# B&R Automation Studio project RS15_RX_30005_r00 (part 5)

#### A1_Control.var - Local variables
```iecst
(********************************************************************
 * COPYRIGHT -- Microsoft
 ********************************************************************
 * Program: A1_Control
 * File: A1_Control.var
 * Author: pkiel
 * Created: July 12, 2011
 ********************************************************************
 * Local variables of program A1_Control
 ********************************************************************)
VAR
  HGW_ChangeReal_0 : HGW_ChangeReal;
  H_RelativeChangeLimitReal1_0 : H_FB_RelativeChangeLimitReal1 ;
  HGW_Toggle_0 : HGW_Toggle;
  HGW_Toggle_1 : HGW_Toggle;
  HMI_FasterPB : BOOL;
  HMI_SlowerPB : BOOL;
  Synch_Permissive : BOOL;
  TOF_0 : TOF;
  bCmd_ManuTimSetPlus  : BOOL ;
  bCmd_ManuTimSetMoins : BOOL ;
  rTemp_ : ARRAY[0..9] OF REAL ;
  rIncrOffsetAxeRun_Inch : REAL ;

  bManuTimSetCond : BOOL ;
  bShiftPerfPos : BOOL ;
  bShiftPerfNeg : BOOL ;
  bEventSelEnvB : BOOL ;

END_VAR
```

- Program Logical/BagMachine_Section/Perf/Axis1/A1_Automat (IEC) - Cam Automat (no source held here)

### Program Logical/BagMachine_Section/Perf/Axis1/A1_Automat2 (IEC) - Cam Automat For Parking Axis

#### A1_Automat2Cyclic.st
```iecst
(********************************************************************
 * COPYRIGHT -- Microsoft
 ********************************************************************
 * Program: A1_Automat2
 * File: A1_Automat2Cyclic.st
 * Author: pkiel
 * Created: July 19, 2011
 ********************************************************************
 * Implementation of program A1_Automat2
 ********************************************************************)

PROGRAM _CYCLIC

(**** CAM AUTOMAT FOR PARKING AXIS ****)
(**** Initialize Automat Parameters Upon Automat Start Request ****)
	Synch_Request := gPerf_ParkRequest;
	IF (Synch_Request AND NOT ParID_Ready) THEN
		MC_BR_InitMasterParIDTransfer_0.Master:=gA[11].Ident;
	    MC_BR_InitMasterParIDTransfer_0.Slave:=gA[1].Ident;
	    MC_BR_InitMasterParIDTransfer_0.MasterParID:=412;
	    MC_BR_InitMasterParIDTransfer_0.SlaveChannel:=0;
	    MC_BR_InitMasterParIDTransfer_0.Execute:=TRUE;
	    IF (MC_BR_InitMasterParIDTransfer_0.Done) THEN
	      MasterParID:=MC_BR_InitMasterParIDTransfer_0.ReceiveParID;
	      MC_BR_InitMasterParIDTransfer_0.Execute:=FALSE;
	      ParID_Ready:=1;
	    ELSIF (MC_BR_InitMasterParIDTransfer_0.Error) THEN
	    (*Store ErrorID in a variable,
	      ErrorID is reset on falling edge of 'Execute'*)
	      ErrorID:=MC_BR_InitMasterParIDTransfer_0.ErrorID;
	      ParID_Ready:=0;
	      MC_BR_InitMasterParIDTransfer_0.Execute:=FALSE;
	    END_IF
	END_IF
	MC_BR_InitMasterParIDTransfer_0();

(**** Initialize Automat Parameters Upon Automat Start Request ****)
  bInitCamAuto := ParID_Ready    AND
                  g_bCameProf_OK AND
                  1              ;

	IF (EDGEPOS(bInitCamAuto))THEN

		(*general automat parameter*)
			AutData.MasterParID		    := MasterParID;
			AutData.StartPosition		:= 0;
			AutData.StartInterval		:= gA[11].AxisPeriod;
			AutData.MaxMasterVelocity	:= gr_rMachMaxSpeed_BPM ;

		(**** Calculations ****)
			gA[1].InchPerDeg := gA[1].UnitsPerDeg/gA[1].UnitsPerInch;
			Travel_Deg := gSP_A[1].ParkPosition-gSP_A[1].MatchedSpeed;
			IF (Travel_Deg<0) THEN
				Travel_Deg := Travel_Deg+360.0;
			END_IF
			Travel_Inch := Travel_Deg*gA[1].InchPerDeg;
			MatchedSpeed_Inch := gSP_A[1].MatchedSpeed*gA[1].InchPerDeg;
			MasterOffset := 0(*gRecipeActive.Perf_Offset*);
			Slave_AxisPeriod := gA[1].AxisPeriod/gSP_PerfKnifeCount;
      rSlave_AxisPeriod_Inch := Slave_AxisPeriod / gA[1].UnitsPerInch ;
      rPosOutMatchedSpeed2_Inch := MatchedSpeed_Inch + rSlave_AxisPeriod_Inch ;

		(**** Slave Starting In Matched Speed Zone ****)
      IF g_bPerfInMatchedSpeed THEN
        InMatched := 1;

			(*Automat STATE 0 Basis State*)
				AutData.State[0].Event[0].Type		:= ncST_END;
				AutData.State[0].Event[0].Attribute	:= ncAT_ONCE;
        AutData.State[0].Event[0].NextState  := 1;

      rTempPosA1_Inch := H_FC_Modulus(IN_rMod:=360*gA[1].InchPerDeg/gSP_PerfKnifeCount, IN_rVar:=gA[1].PositionInch) ;

			(*Initial Matched Speed Zone*)
				AutData.State[1].CamProfileIndex	:= 16#FFFF;
				AutData.State[1].MasterFactor		:= REAL_TO_UDINT((MatchedSpeed_Inch-rTempPosA1_Inch)*gA[11].UnitsPerInch);
				AutData.State[1].SlaveFactor		:= REAL_TO_DINT((MatchedSpeed_Inch-rTempPosA1_Inch)*gA[1].UnitsPerInch);
				AutData.State[1].CompMode			:= ncOFF;

				AutData.State[1].Event[0].Type		:= ncST_END;
				AutData.State[1].Event[0].Attribute	:= ncST_END;
				AutData.State[1].Event[0].NextState	:= 2;

			(*Initial Comp With Matched Speed Zone*)
				AutData.State[2].CamProfileIndex	:= 16#FFFF;
				AutData.State[2].MasterFactor		:= REAL_TO_UDINT(MatchedSpeed_Inch*gA[11].UnitsPerInch);
				AutData.State[2].SlaveFactor		:= REAL_TO_DINT(MatchedSpeed_Inch*gA[1].UnitsPerInch);
				AutData.State[2].CompMode			:= ncONLYCOMP;
				AutData.State[2].MasterCompDistance	:= (gA[11].AxisPeriod)-((gA[11].PositionInch+MasterOffset)*gA[11].UnitsPerInch)-AutData.State[1].MasterFactor;
				AutData.State[2].SlaveCompDistance	:= (Slave_AxisPeriod)-gA[1].PositionCount-AutData.State[1].SlaveFactor;

				IF (AutData.State[2].SlaveCompDistance<=0) THEN
					AutData.State[2].SlaveCompDistance := AutData.State[2].SlaveCompDistance+Slave_AxisPeriod;
				END_IF
				IF (AutData.State[2].MasterCompDistance<0) THEN
					Value1 := REAL_TO_DINT(AutData.State[2].MasterCompDistance*1000.0);
					Value2 := REAL_TO_DINT(gA[11].AxisPeriod*1000.0);
					AutData.State[2].MasterCompDistance := (DINT_TO_REAL(Value1 MOD Value2))/1000.0;
					IF (AutData.State[2].MasterCompDistance<0) THEN
						AutData.State[2].MasterCompDistance := AutData.State[2].MasterCompDistance+gA[11].AxisPeriod;
					END_IF
				END_IF
				IF ((AutData.State[2].MasterCompDistance<(0.5*gA[11].AxisPeriod)) AND (AutData.State[2].SlaveCompDistance>(0.5*Slave_AxisPeriod))) THEN
					AutData.State[2].MasterCompDistance := AutData.State[2].MasterCompDistance+(gA[11].AxisPeriod);
				END_IF
				IF (AutData.State[2].MasterCompDistance<(0.1*gA[11].AxisPeriod)) THEN
					AutData.State[2].MasterCompDistance := AutData.State[2].MasterCompDistance+(gA[11].AxisPeriod);
				END_IF

				AutData.State[2].Event[0].Type		:= ncST_END;
				AutData.State[2].Event[0].Attribute	:= ncST_END;
				AutData.State[2].Event[0].NextState	:= 3;

			ELSE
				InMatched := 0;

			(*Automat STATE 0 Basis State*)
				AutData.State[0].Event[0].Type		:= ncST_END;
				AutData.State[0].Event[0].Attribute	:= ncAT_ONCE;
				AutData.State[0].Event[0].NextState	:= 2;

			(*Initial Matched Speed Zone...NOT USED*)
				AutData.State[1].CamProfileIndex	:= 16#FFFE;
				AutData.State[1].MasterFactor		:= 1;
				AutData.State[1].SlaveFactor		:= 1;
				AutData.State[1].CompMode			:= ncOFF;

				AutData.State[1].Event[0].Type		:= ncST_END;
				AutData.State[1].Event[0].Attribute	:= ncST_END;
				AutData.State[1].Event[0].NextState	:= 3;

			(*Initial Comp With Matched Speed Zone*)
				AutData.State[2].CamProfileIndex	:= 16#FFFF;
				AutData.State[2].MasterFactor		:= REAL_TO_UDINT(MatchedSpeed_Inch*gA[11].UnitsPerInch);
				AutData.State[2].SlaveFactor		:= REAL_TO_DINT(MatchedSpeed_Inch*gA[1].UnitsPerInch);
				AutData.State[2].CompMode			:= ncONLYCOMP;
				AutData.State[2].MasterCompDistance	:= gA[11].AxisPeriod-((gA[11].PositionInch+MasterOffset)*gA[11].UnitsPerInch);
				AutData.State[2].SlaveCompDistance	:= Slave_AxisPeriod-gA[1].PositionCount;

				IF (AutData.State[2].SlaveCompDistance<=0) THEN
					AutData.State[2].SlaveCompDistance := AutData.State[2].SlaveCompDistance+Slave_AxisPeriod;
				END_IF
				IF (AutData.State[2].MasterCompDistance<0) THEN
					Value1 := REAL_TO_DINT(AutData.State[2].MasterCompDistance*1000.0);
					Value2 := REAL_TO_DINT(gA[11].AxisPeriod*1000.0);
					AutData.State[2].MasterCompDistance := (DINT_TO_REAL(Value1 MOD Value2))/1000.0;
					IF (AutData.State[2].MasterCompDistance<0) THEN
						AutData.State[2].MasterCompDistance := AutData.State[2].MasterCompDistance+gA[11].AxisPeriod;
					END_IF
				END_IF
				IF ((AutData.State[2].MasterCompDistance<(0.5*gA[11].AxisPeriod)) AND (AutData.State[2].SlaveCompDistance>(0.5*Slave_AxisPeriod))) THEN
					AutData.State[2].MasterCompDistance := AutData.State[2].MasterCompDistance+(gA[11].AxisPeriod);
				END_IF
				IF (AutData.State[2].MasterCompDistance<(0.1*gA[11].AxisPeriod)) THEN
					AutData.State[2].MasterCompDistance := AutData.State[2].MasterCompDistance+(gA[11].AxisPeriod);
				END_IF

				AutData.State[2].Event[0].Type		:= ncST_END;
				AutData.State[2].Event[0].Attribute	:= ncST_END;
				AutData.State[2].Event[0].NextState	:= 3;

			END_IF

		(*Running Comp With Matched Speed Zone *)
			AutData.State[3].CamProfileIndex	:= 16#FFFE;
			AutData.State[3].MasterFactor		:= 1;
			AutData.State[3].SlaveFactor		:= 0;
			AutData.State[3].CompMode			:= ncONLYCOMP;
			AutData.State[3].MasterCompDistance	:= Travel_Inch*gA[11].UnitsPerInch;
			AutData.State[3].SlaveCompDistance	:= Travel_Inch*gA[1].UnitsPerInch;

			AutData.State[3].Event[0].Type		:= ncST_END;
			AutData.State[3].Event[0].Attribute	:= ncST_END;
			AutData.State[3].Event[0].NextState	:= 4;

		(*Running Comp With Matched Speed Zone *)
			AutData.State[4].CamProfileIndex	:= 16#FFFF;
			AutData.State[4].MasterFactor		:= REAL_TO_UDINT(Slave_AxisPeriod);
			AutData.State[4].SlaveFactor		:= 0;
			AutData.State[4].CompMode			:= ncOFF;

			AutData.State[4].Event[0].Type		:= ncST_END;
			AutData.State[4].Event[0].Attribute	:= ncST_END;
			AutData.State[4].Event[0].NextState	:= 4;

		(*Initialize & Enable the Automat Control *)
			MC_BR_AutControl_0.Enable 		:= 1;
			MC_BR_AutControl_0.AdrAutData 	:= ADR(AutData);
			MC_BR_AutControl_0.InitAutData 	:= 1;
	END_IF
		(* wait for initialization done*)
			IF ((MC_BR_AutControl_0.AutDataInitialized = 1) AND (Synch_Request)) THEN
				MC_BR_AutControl_0.InitAutData 	:= 0;
				AutomatStart := 1;
			END_IF
			(* check if error occured *)
			IF (MC_BR_AutControl_0.ErrorID <> 0) THEN
				Error := MC_BR_AutControl_0.ErrorID;
				MC_BR_AutControl_0.Enable := 0;
			END_IF

	(******************** ENABLE CAM-AUTOMAT **********************)

	IF (AutomatStart) THEN
			MC_BR_AutControl_0.Start := 1;
			AutomatStart := 0;
	END_IF

	IF (NOT Synch_Request) THEN
			MC_BR_AutControl_0.Stop := 1;
			MC_BR_AutControl_0.Start := 0;
			ParID_Ready := 0;
			IF (MC_BR_AutControl_0.Running=0) THEN
				MC_BR_AutControl_0.Enable := 0;
				MC_BR_AutControl_0.Stop := 0;
			END_IF
	END_IF

	IF (gPerf_ParkRequired) THEN
		gA[1].Ind_AutomatEnabled:=MC_BR_AutControl_0.Enable;
		gA[1].Ind_CurrentAutomatState:=MC_BR_AutControl_0.ActualStateIndex;
	END_IF

	(********************** MC_AUTCONTROL *************************)
	MC_BR_AutControl_0.Slave:= gA[1].Ident;
	MC_BR_AutControl_0();

END_PROGRAM
```

### Program Logical/BagMachine_Section/Perf/Axis1/A1_Ref (IEC) - Reference Routine

#### A1_Ref.var - Local variables
```iecst
(********************************************************************
 * COPYRIGHT -- Microsoft
 ********************************************************************
 * Program: A1_Ref
 * File: A1_Ref.var
 * Author: pkiel
 * Created: July 13, 2011
 ********************************************************************
 * Local variables of program A1_Ref
 ********************************************************************)
VAR
	HGW_2StateIND_0 : HGW_2StateIND;
	HGW_2StepMove_0 : HGW_2StepMove;
	MC_Home_0 : MC_Home;
	RefPBColor_Ind : UINT;
END_VAR
```

### Program Logical/BagMachine_Section/Perf/Axis1/A1_Cycle (IEC) - A new program

#### A1_CycleCyclic.st
```iecst
(********************************************************************
 * COPYRIGHT -- .
 ********************************************************************
 * Program: A1_Cycle
 * File: A1_CycleCyclic.st
 * Author: dominique
 * Created: August 01, 2011
 ********************************************************************
 * Implementation of program A1_Cycle
 ********************************************************************)

PROGRAM _CYCLIC

// Manu axis movement for timing setting

    //---------------------------------------------------------------------------------------------------------------------
    // ACDC Power Supply cycle
    //---------------------------------------------------------------------------------------------------------------------
    // Start cycle
    gstCycA[1].CycManTimSet.CmdStart := ( gA[1].Cmd_ManuTimSetPlus    OR
                                          gA[1].Cmd_ManuTimSetMinus ) AND
                                        NOT(gA[1].Error)              AND
                                        NOT(gA[11].Error)             ;
    IF gstCycA[1].CycManTimSet.CmdStart THEN
      gstCycA[1].CycManTimSet.bSCyc := 1 ;
    END_IF ;

    //----------------------------------------------------------------------
    // Cycle at rest
    IF NOT(gstCycA[1].CycManTimSet.bSCyc) AND
       1                                 THEN
      IF NOT( gstCycA[1].CycManTimSet.bFCyc ) THEN
        // Init after cycle unpropaly ended
        gstCycA[1].CycManTimSet.bFCyc := 1 ;
        gstCycA[1].CycManTimSet.bCyc  := 0 ;

        gstCycA[1].CycManTimSet.CmdMov  := 0 ;
        gstCycA[1].CycManTimSet.CmdStop := 0 ;
        gstCycA[1].CycManTimSet.CmdSynchroOn := 0 ;
      END_IF
      gstCycA[1].CycManTimSet.iStep := 0 ;
      RETURN ;
    ELSE
    //----------------------------------------------------------------------
    // Cycle running

      // Permanent conditions
      IF NOT(gA[1].Ind_Ready)                  OR
         NOT(gA[11].Ind_Ready)                 OR
         NOT(gstCycA[1].CycManTimSet.CmdStart) AND
         (gstCycA[1].CycManTimSet.iStep <= 2)  THEN
        gstCycA[1].CycManTimSet.bSCyc := 0 ;
        RETURN ;
      END_IF

      // Permanent actions
      stTON_01 (
            IN := ( gstCycA[1].CycManTimSet.iStep = C_iSTEP_0 ) ,
            PT := T#30ms
               ) ;
    END_IF
    //----------------------------------------------------------------------
    // Cycle steps

        CASE gstCycA[1].CycManTimSet.iStep OF

        C_iSTEP_0 :
         //----------------------------------------------
         // Etape 1 : Initialisation
         //----------------------------------------------
          IF stTON_01.Q THEN
            gstCycA[1].CycManTimSet.iStep := C_iSTEP_1 ;

            // Action Step 1
            gstCycA[1].CycManTimSet.bFCyc := 0 ;
            gstCycA[1].CycManTimSet.bCyc  := 1 ;
          END_IF

        C_iSTEP_1 :
         //----------------------------------------------
         // Etape 2 : Synchro Drum
         //----------------------------------------------
          IF TRUE THEN
            gstCycA[1].CycManTimSet.iStep := C_iSTEP_2 ;

            // Action Step 2
            gstCycA[1].CycManTimSet.CmdSynchroOn := 1 ;
          END_IF

        C_iSTEP_2 :
         //----------------------------------------------
         // Step 3 : Activation motion and Stop waiting
         //----------------------------------------------
          IF gstCycA[1].CycManTimSet.bSynchroOkSlavA[11] THEN
            gstCycA[1].CycManTimSet.iStep := C_iSTEP_3 ;

            // Action Step 3
            gstCycA[1].CycManTimSet.CmdMov  := 1 ;
            gstCycA[1].CycManTimSet.CmdStop := 0 ;
            // Stop waiting
          END_IF

        C_iSTEP_3 :
         //----------------------------------------------
         // Step 4 : Stop motion and End stop waiting
         //----------------------------------------------
          IF NOT(gstCycA[1].CycManTimSet.CmdStart) THEN
            gstCycA[1].CycManTimSet.iStep := C_iSTEP_4 ;

            // Action Step 4
            gstCycA[1].CycManTimSet.CmdMov  := 0 ;
            gstCycA[1].CycManTimSet.CmdStop := 1 ;
            // End stop waiting
          END_IF

        C_iSTEP_4 :
         //----------------------------------------------
         // Step 3 : Activation motion and Stop waiting
         // Step 5 : Cut synchro
         //----------------------------------------------
          // Condition Step3
          IF gstCycA[1].CycManTimSet.CmdStart THEN
            gstCycA[1].CycManTimSet.iStep := C_iSTEP_3 ;

            // Action Step 3
            gstCycA[1].CycManTimSet.CmdMov  := 1 ;
            gstCycA[1].CycManTimSet.CmdStop := 0 ;
            // Stop waiting
            RETURN ;
          END_IF ;
          // Condition Step5
          IF NOT(gstCycA[1].CycManTimSet.CmdStop) THEN
            gstCycA[1].CycManTimSet.iStep := C_iSTEP_5 ;

            // Action Step 5
            gstCycA[1].CycManTimSet.CmdSynchroOn := 0 ;
          END_IF

        C_iSTEP_5 :
         //----------------------------------------------
         // Step 6 : New offset calculation
         //----------------------------------------------
          IF TRUE THEN
            gstCycA[1].CycManTimSet.iStep := C_iSTEP_6 ;

            // Action Step 6
            // Memo Actual phase Offset
            rTempActPhasDeg[1]    := gRecipeActive.rPerf_PhasMasterDeg ;
            rTempActOffsetInch[1] := gRecipeActive.Perf_Offset ;
            // Update phase
            gRecipeActive.rPerf_PhasMasterDeg := gA[11].rActPhasDeg ;
            // Update Offset
            rTemp_[1] := gA[11].PositionInch - gA[9].PositionInch ;
            gRecipeActive.Perf_Offset := H_FC_Modulus (IN_rMod := gRecipeActive.Repeat, IN_rVar := rTemp_[1]) ;
          END_IF

        C_iSTEP_6 :
         //----------------------------------------------
         // Step 0 : First step
         //----------------------------------------------
          IF TRUE THEN
            gstCycA[1].CycManTimSet.iStep := C_iSTEP_0 ;

            // Action Step 0
            gstCycA[1].CycManTimSet.bSCyc := 0 ;
            gstCycA[1].CycManTimSet.bFCyc := 1 ;
            gstCycA[1].CycManTimSet.bCyc  := 0 ;
          END_IF
        END_CASE
    //---------------------------------------------------------------------------------------------------------------------

END_PROGRAM
```

### Program Logical/BagMachine_Section/Perf/Axis1/A1_CamProfCalc (IEC) - A new program

#### A1_CamProfCalcInit.st - Initialization code
```iecst
(********************************************************************
 * COPYRIGHT -- .
 ********************************************************************
 * Program: A1_CamProfCalc
 * File: A1_CamProfCalcInit.st
 * Author: dominique
 * Created: August 24, 2011
 ********************************************************************
 * Implementation of program A1_CamProfCalc
 ********************************************************************)

PROGRAM _INIT
  // Came profile Perf index
  g_uiIndexCamProfPerf := 1 ;

END_PROGRAM
```

### Program Logical/BagMachine_Section/Perf/Axis11_VirtualAxis/A11_Automat

#### A11_AutomatCyclic.st
```iecst
(********************************************************************
 * COPYRIGHT -- Microsoft
 ********************************************************************
 * Program: A11_Automat
 * File: A11_AutomatCyclic.st
 * Author: pkiel
 * Created: July 22, 2011
 ********************************************************************
 * Implementation of program A11_Automat
 ********************************************************************)

PROGRAM _CYCLIC

  // Synchro ratio Master/Slave
     // Master = Virtuel
     gA[11].rRSynNum := 1 ;
     gA[11].rRSynDen := 1 ;

  // Signal synchro Holding axis
  MC_BR_AutControl_0.Signal1 := gA[3].Ind_bSynchroOK ;

  // Perf  manu moving
  MC_BR_AutControl_0.Signal2 := 0 ;

  IF gstCycA[1].CycManTimSet.CmdSynchroOn THEN
    MC_BR_AutControl_0.Signal2 := 1 ;
  END_IF

  // A11 Synchro OK indicator
  gstCycA[1].CycManTimSet.bSynchroOkSlavA[11] := ( MC_BR_AutControl_0.ActualStateIndex = 3 )   AND
                                                 gA[11].Ind_SynchronizedMotion AND ParID_Ready ;

(**** STRAIGHT GEARED CAM AUTOMAT WITH ABSOLUTE PHASE SYNCHRONIZATION FOR TEARING AXIS ***)

(* Set Up Master Position Parameter ID *)
  Synch_Request := gA[11].Cmd_SynchronizedMotion;
  IF (Synch_Request AND NOT ParID_Ready) THEN
    MC_BR_InitMasterParIDTransfer_0.Master:=gA[9].Ident;
      MC_BR_InitMasterParIDTransfer_0.Slave:=gA[11].Ident;
      MC_BR_InitMasterParIDTransfer_0.MasterParID:=412;   // 412: VAX: Position, S_SET_VAX1, DINT
      MC_BR_InitMasterParIDTransfer_0.SlaveChannel:=0;
      MC_BR_InitMasterParIDTransfer_0.Execute:=TRUE;
      IF (MC_BR_InitMasterParIDTransfer_0.Done) THEN
        MasterParID:=MC_BR_InitMasterParIDTransfer_0.ReceiveParID;
        MC_BR_InitMasterParIDTransfer_0.Execute:=FALSE;
        ParID_Ready:=1;
      ELSIF (MC_BR_InitMasterParIDTransfer_0.Error) THEN
      (*Store ErrorID in a variable,
        ErrorID is reset on falling edge of 'Execute'*)
        ErrorID:=MC_BR_InitMasterParIDTransfer_0.ErrorID;
        ParID_Ready:=0;
        MC_BR_InitMasterParIDTransfer_0.Execute:=FALSE;
      END_IF
  END_IF
  MC_BR_InitMasterParIDTransfer_0();

(**** Initialize Automat Parameters Upon Automat Start Request ****)
  IF (EDGEPOS(ParID_Ready AND g_bCameProf_OK))THEN

    (**** Calculate Slave Start Offset ****)
      PositionOffset:= REAL_TO_DINT((gA[9].PositionInch-(gA[11].PositionInch-gRecipeActive.Perf_Offset))*1000);
      PositionMOD:= REAL_TO_DINT(gRecipeActive.Repeat*1000);
      SlaveStartOffset:= (DINT_TO_REAL(PositionOffset MOD PositionMOD))/1000;
      IF (SlaveStartOffset >= (0.5*gRecipeActive.Repeat)) THEN
        SlaveStartOffset := SlaveStartOffset - gRecipeActive.Repeat;
      END_IF
      IF (SlaveStartOffset < (-0.5*gRecipeActive.Repeat)) THEN
        SlaveStartOffset := SlaveStartOffset + gRecipeActive.Repeat;
      END_IF

      MasterOffset := gRecipeActive.Perf_Offset ;
      MatchedSpeed_Inch := gSP_A[1].MatchedSpeed * gA[1].InchPerDeg ;

    (*general automat parameter*)
      AutData.MasterParID        := MasterParID;
      AutData.StartPosition      := 0;
      AutData.StartInterval      := gA[9].AxisPeriod;
      AutData.MaxMasterVelocity  := gr_rMachMaxSpeed_BPM ;

    (*Automat STATE 0 Basis State*)
      AutData.State[0].Event[0].Type    := ncST_END;
      AutData.State[0].Event[0].Attribute  := ncAT_ONCE;
      //AutData.State[0].Event[0].NextState  := 1;
      AutData.State[0].Event[0].NextState  := 10;

    //Waiting synchro Holding axis
      AutData.State[10].CamProfileIndex := 16#FFFF;
      AutData.State[10].MasterFactor    := REAL_TO_UDINT(gA[9].AxisPeriod);
      AutData.State[10].SlaveFactor     := 0;
      AutData.State[10].CompMode        := ncOFF;

      AutData.State[10].Event[1].Type      := ncSIGNAL2 ;
      AutData.State[10].Event[1].Attribute := ncAT_ONCE ;
      AutData.State[10].Event[1].NextState := 3 ;

    //**** Slave Starting In Matched Speed Zone ***
      IF g_bPerfInMatchedSpeed THEN
        InMatched := 1;

      //Automat STATE 0 Basis State
        AutData.State[10].Event[0].Type      := ncSIGNAL1;
        AutData.State[10].Event[0].Attribute := ncAT_ONCE;
        AutData.State[10].Event[0].NextState := 1;

        rTempPosA1_Inch := H_FC_Modulus(IN_rMod:=360*gA[1].InchPerDeg/gSP_PerfKnifeCount, IN_rVar:=gA[1].PositionInch) ;

      //Initial Matched Speed Zone
        AutData.State[1].CamProfileIndex := 16#FFFF;
        AutData.State[1].MasterFactor    := REAL_TO_UDINT((MatchedSpeed_Inch-rTempPosA1_Inch)*gA[9].UnitsPerInch);
        AutData.State[1].SlaveFactor     := REAL_TO_UDINT((MatchedSpeed_Inch-rTempPosA1_Inch)*gA[11].UnitsPerInch);
        AutData.State[1].CompMode        := ncOFF;

        AutData.State[1].Event[0].Type      := ncST_END ;
        AutData.State[1].Event[0].Attribute := ncST_END;
        AutData.State[1].Event[0].NextState := 2;

        AutData.State[1].Event[1].Type      := ncSIGNAL2 ;
        AutData.State[1].Event[1].Attribute := ncAT_ONCE ;
        AutData.State[1].Event[1].NextState := 3 ;

      //Initial Comp With Matched Speed Zone
        AutData.State[2].CamProfileIndex    := 16#FFFF;
        AutData.State[2].MasterFactor       := REAL_TO_UDINT(MatchedSpeed_Inch*gA[9].UnitsPerInch);
        AutData.State[2].SlaveFactor        := REAL_TO_UDINT(MatchedSpeed_Inch*gA[11].UnitsPerInch);
        AutData.State[2].CompMode           := ncONLYCOMP;
        AutData.State[2].MasterCompDistance := (gA[9].AxisPeriod)-((gA[9].PositionInch+MasterOffset)*gA[9].UnitsPerInch)-AutData.State[1].MasterFactor;
        AutData.State[2].SlaveCompDistance  := (gA[11].AxisPeriod)-gA[11].PositionCount-AutData.State[1].SlaveFactor;

        IF (AutData.State[2].SlaveCompDistance<=0) THEN
          AutData.State[2].SlaveCompDistance := AutData.State[2].SlaveCompDistance+gA[11].AxisPeriod;
        END_IF
        IF (AutData.State[2].MasterCompDistance<0) THEN
          Value1 := REAL_TO_DINT(AutData.State[2].MasterCompDistance);
          Value2 := REAL_TO_DINT(gA[9].AxisPeriod);
          AutData.State[2].MasterCompDistance := DINT_TO_REAL(Value1 MOD Value2);
          IF (AutData.State[2].MasterCompDistance<0) THEN
            AutData.State[2].MasterCompDistance := AutData.State[2].MasterCompDistance+gA[9].AxisPeriod;
          END_IF
        END_IF

        IF ((AutData.State[2].MasterCompDistance<(0.5*gA[9].AxisPeriod)) AND (AutData.State[2].SlaveCompDistance>(0.5*gA[11].AxisPeriod))) THEN
          AutData.State[2].MasterCompDistance := AutData.State[2].MasterCompDistance+(gA[9].AxisPeriod);
        END_IF

        AutData.State[2].Event[0].Type      := ncST_END ;
        AutData.State[2].Event[0].Attribute := ncST_END;
        AutData.State[2].Event[0].NextState := 3;

        AutData.State[2].Event[1].Type      := ncSIGNAL2 ;
        AutData.State[2].Event[1].Attribute := ncAT_ONCE ;
        AutData.State[2].Event[1].NextState := 3 ;

      ELSE
        InMatched := 0;

      //Automat STATE 0 Basis State
        AutData.State[10].Event[0].Type       := ncSIGNAL1;
        AutData.State[10].Event[0].Attribute  := ncAT_ONCE;
        AutData.State[10].Event[0].NextState  := 5 ;

      //Initial Comp With Matched Speed Zone
        AutData.State[5].CamProfileIndex    := 16#FFFF;
        AutData.State[5].MasterFactor       := REAL_TO_UDINT(MatchedSpeed_Inch*gA[9].UnitsPerInch);
        AutData.State[5].SlaveFactor        := REAL_TO_UDINT(MatchedSpeed_Inch*gA[11].UnitsPerInch);
        AutData.State[5].CompMode           := ncONLYCOMP;
        AutData.State[5].MasterCompDistance := gA[9].AxisPeriod-((gA[9].PositionInch+MasterOffset)*gA[9].UnitsPerInch);
        AutData.State[5].SlaveCompDistance  := gA[11].AxisPeriod-gA[11].PositionCount;

        IF (AutData.State[5].SlaveCompDistance<=0) THEN
          AutData.State[5].SlaveCompDistance := AutData.State[5].SlaveCompDistance+gA[11].AxisPeriod;
        END_IF
        IF (AutData.State[5].MasterCompDistance<0) THEN
          Value1 := REAL_TO_DINT(AutData.State[5].MasterCompDistance);
          Value2 := REAL_TO_DINT(gA[9].AxisPeriod);
          AutData.State[5].MasterCompDistance := DINT_TO_REAL(Value1 MOD Value2);
          IF (AutData.State[5].MasterCompDistance<0) THEN
            AutData.State[5].MasterCompDistance := AutData.State[5].MasterCompDistance+gA[9].AxisPeriod;
          END_IF
        END_IF

        IF ((AutData.State[5].MasterCompDistance<(0.5*gA[9].AxisPeriod)) AND (AutData.State[5].SlaveCompDistance>(0.5*gA[11].AxisPeriod))) THEN
          AutData.State[5].MasterCompDistance := AutData.State[5].MasterCompDistance+(gA[9].AxisPeriod);
        END_IF

        AutData.State[5].Event[0].Type      := ncST_END ;
        AutData.State[5].Event[0].Attribute := ncST_END;
        AutData.State[5].Event[0].NextState := 3;

        AutData.State[5].Event[1].Type      := ncSIGNAL2 ;
        AutData.State[5].Event[1].Attribute := ncAT_ONCE ;
        AutData.State[5].Event[1].NextState := 3 ;

      END_IF

    (*Automat STATE 3 Master/Slave Run*)
      AutData.State[3].CamProfileIndex   := 16#FFFF;
      AutData.State[3].MasterFactor      := REAL_TO_UDINT(gA[9].AxisPeriod);
      AutData.State[3].SlaveFactor       := REAL_TO_UDINT(gA[11].AxisPeriod);
      AutData.State[3].CompMode          := ncOFF;

      AutData.State[3].Event[0].Type       := ncST_END;
      AutData.State[3].Event[0].Attribute  := ncST_END;
      AutData.State[3].Event[0].NextState  := 3;

      MC_BR_AutControl_0.Enable       := 1;
      MC_BR_AutControl_0.AdrAutData   := ADR(AutData);
      MC_BR_AutControl_0.InitAutData  := 1;
  END_IF
      (* wait for initialization done or restart *)
      IF ((MC_BR_AutControl_0.AutDataInitialized=1) AND (Synch_Request)) THEN
        MC_BR_AutControl_0.InitAutData := 0;
        MC_BR_AutControl_0.Enable :=1;
        AutomatStart := 1;;
      END_IF
      (* check if error occured *)
      IF (MC_BR_AutControl_0.ErrorID <> 0) THEN
        MC_BR_AutControl_0.Enable := 0;
      END_IF

  (******************** ENABLE CAM-AUTOMAT **********************)

  IF (AutomatStart) THEN
      MC_BR_AutControl_0.Start := 1;
      AutomatStart := 0;
  END_IF

  IF (NOT Synch_Request) THEN
      MC_BR_AutControl_0.Stop := 1;
      MC_BR_AutControl_0.Start := 0;
      ParID_Ready := 0;
      IF (MC_BR_AutControl_0.Running=0) THEN
        MC_BR_AutControl_0.Enable := 0;
        MC_BR_AutControl_0.Stop := 0;
      END_IF
  END_IF

  gA[11].Ind_AutomatEnabled:=MC_BR_AutControl_0.Enable;
  gA[11].Ind_CurrentAutomatState:=MC_BR_AutControl_0.ActualStateIndex;
  gA[11].Ind_bSynchroOK := (MC_BR_AutControl_0.ActualStateIndex = 3) AND gA[11].Ind_SynchronizedMotion ;

  (********************** MC_AUTCONTROL *************************)
  MC_BR_AutControl_0.Slave:= gA[11].Ident;
  MC_BR_AutControl_0();

END_PROGRAM
```

- Program Logical/BagMachine_Section/Perf/Axis11_VirtualAxis/A11_Basic (IEC) (no source held here)

### Program Logical/BagMachine_Section/Perf/Axis11_VirtualAxis/A11_Control

#### A11_Control.var
```iecst
(********************************************************************
 * COPYRIGHT -- Microsoft
 ********************************************************************
 * Program: A11_Control
 * File: A11_Control.var
 * Author: pkiel
 * Created: July 22, 2011
 ********************************************************************
 * Local variables of program A11_Control
 ********************************************************************)
VAR
	HGW_ChangeReal_0 : HGW_ChangeReal;
  H_RelativeChangeLimitReal1_0 : H_FB_RelativeChangeLimitReal1 ;
	HGW_Toggle_0 : HGW_Toggle;
	HGW_Toggle_1 : HGW_Toggle;
	HMI_FasterPB : BOOL;
	HMI_SlowerPB : BOOL;
	Synch_Permissive : BOOL;
	TOF_0 : TOF;
  bCmd_ManuTimSetPlus  : BOOL ;
  bCmd_ManuTimSetMoins : BOOL ;
  rTemp_ : ARRAY[0..9] OF REAL ;
  rIncrOffsetAxeRun_Inch : REAL ;

END_VAR
```

#### A11_ControlCyclic.ld
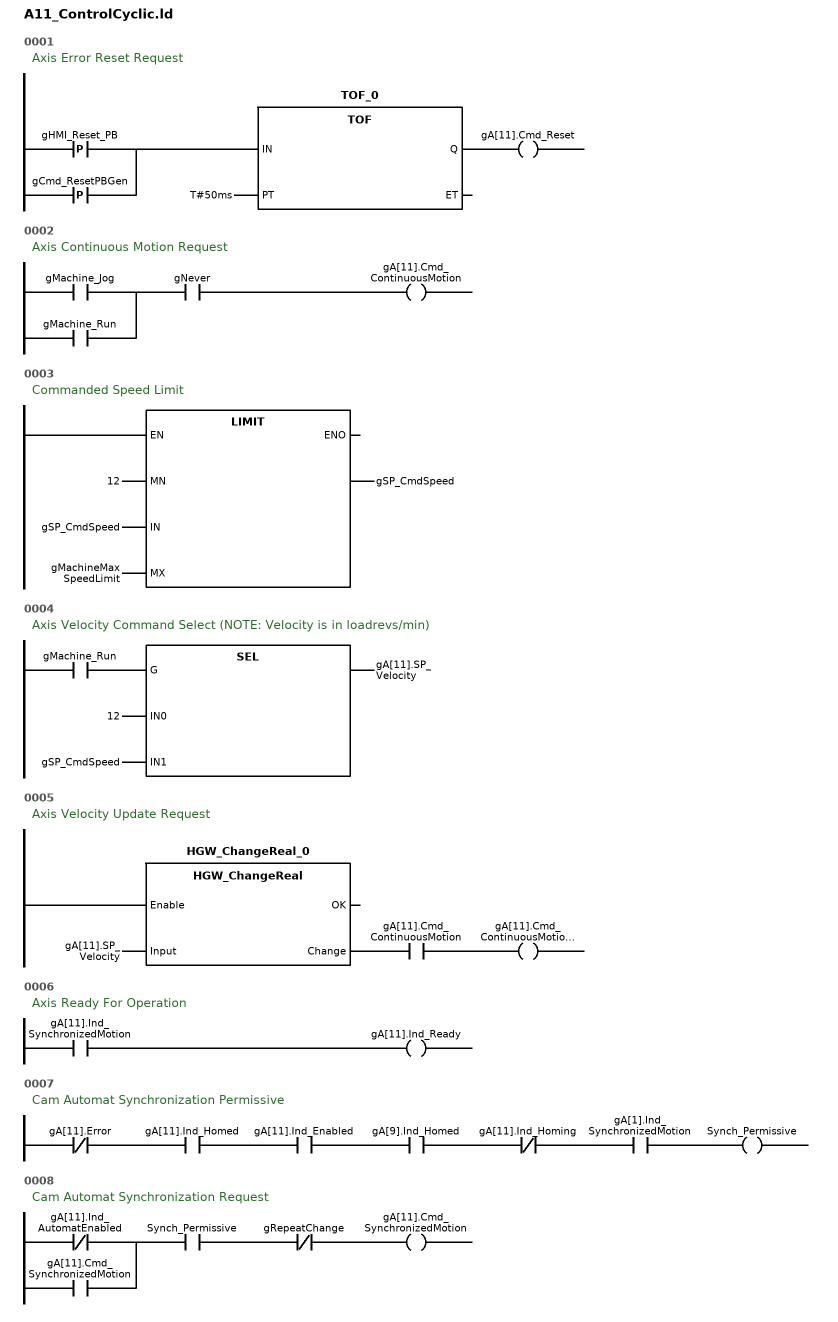
Ladder, written as Structured Text:
```iecst
(********************************************************************
 * COPYRIGHT -- Microsoft
 ********************************************************************
 * Program: A11_Control
 * File: A11_ControlCyclic.ld
 * Author: pkiel
 * Created: July 22, 2011
 ********************************************************************
 * Implementation of program A11_Control
 ********************************************************************)

PROGRAM _CYCLIC
VAR
    _e1 : R_TRIG;
    _e2 : R_TRIG;
END_VAR
(* Network 1: Axis Error Reset Request *)
_e1(CLK := gHMI_Reset_PB);
_e2(CLK := gCmd_ResetPBGen);
TOF_0(IN := _e1.Q OR _e2.Q, PT := T#50ms);
gA[11].Cmd_Reset := TOF_0.Q;

(* Network 2: Axis Continuous Motion Request *)
gA[11].Cmd_ContinuousMotion := (gMachine_Jog OR gMachine_Run) AND gNever;

(* Network 3: Commanded Speed Limit *)
gSP_CmdSpeed := LIMIT(MN := 12, IN := gSP_CmdSpeed, MX := gMachineMaxSpeedLimit);

(* Network 4: Axis Velocity Command Select (NOTE: Velocity is in loadrevs/min) *)
gA[11].SP_Velocity := SEL(G := gMachine_Run, IN0 := 12, IN1 := gSP_CmdSpeed);

(* Network 5: Axis Velocity Update Request *)
HGW_ChangeReal_0(Enable := TRUE, Input := gA[11].SP_Velocity);
gA[11].Cmd_ContinuousMotionUpdate := HGW_ChangeReal_0.Change AND gA[11].Cmd_ContinuousMotion;

(* Network 6: Axis Ready For Operation *)
gA[11].Ind_Ready := gA[11].Ind_SynchronizedMotion;

(* Network 7: Cam Automat Synchronization Permissive *)
Synch_Permissive := NOT gA[11].Error AND gA[11].Ind_Homed AND gA[11].Ind_Enabled AND gA[9].Ind_Homed AND NOT gA[11].Ind_Homing AND gA[1].Ind_SynchronizedMotion;

(* Network 8: Cam Automat Synchronization Request *)
gA[11].Cmd_SynchronizedMotion := (NOT gA[11].Ind_AutomatEnabled OR gA[11].Cmd_SynchronizedMotion) AND Synch_Permissive AND NOT gRepeatChange;
END_PROGRAM
```

- A11_Initl.vax (not shown)

### A11_Par.apt
```
AcoposParameterTable:
  Root Parameters:
    110 = ncSW_OFF (Name=CMD_SIMULATION)  // Simulation mode: Command
    128 = 1 (Name=SGEN_SW_END_IGNORE)  // SGEN_SW_END_IGNORE
```

### Program Logical/BagMachine_Section/RS_Glue

#### RS_GlueCyclic.st
```iecst
(********************************************************************
 * COPYRIGHT -- Microsoft
 ********************************************************************
 * Program: RS_Glue
 * File: RS_GlueCyclic.st
 * Author: dominique
 * Created: October 26, 2011
 ********************************************************************
 * Implementation of program ColdGlue
 ********************************************************************)

PROGRAM _CYCLIC
  // Limit operator setpoint
  gSP_RSGlue.MinPressure := LIMIT (0,gSP_RSGlue.MinPressure,399) ;
  gSP_RSGlue.MaxPressure := LIMIT (0,gSP_RSGlue.MaxPressure,400) ;

  // Type RS glue selection (Cold/Hot)
  gQ_CR_HotColdRSGlueSelect := gRecipeActive.bSelTypeRSGlue ;
  IF EDGEPOS(gRecipeActive.bSelTypeRSGlue) THEN
    // Switch set points on screen from Cold to Hot
    stSP_ColdGlue.MinPressure := gSP_RSGlue.MinPressure ;
    stSP_ColdGlue.MaxPressure := gSP_RSGlue.MaxPressure ;
    stSP_ColdGlue.ManPressure := gSP_RSGlue.ManPressure ;
    stSP_ColdGlue.AutoOnSpeed := gSP_RSGlue.AutoOnSpeed ;

    gSP_RSGlue.MinPressure := stSP_HotGlue.MinPressure ;
    gSP_RSGlue.MaxPressure := stSP_HotGlue.MaxPressure ;
    gSP_RSGlue.ManPressure := stSP_HotGlue.ManPressure ;
    gSP_RSGlue.AutoOnSpeed := stSP_HotGlue.AutoOnSpeed ;
  END_IF ;
  IF EDGENEG(gRecipeActive.bSelTypeRSGlue) THEN
    // Switch set points on screen from Hot to Cold
    stSP_HotGlue.MinPressure := gSP_RSGlue.MinPressure ;
    stSP_HotGlue.MaxPressure := gSP_RSGlue.MaxPressure ;
    stSP_HotGlue.ManPressure := gSP_RSGlue.ManPressure ;
    stSP_HotGlue.AutoOnSpeed := gSP_RSGlue.AutoOnSpeed ;

    gSP_RSGlue.MinPressure := stSP_ColdGlue.MinPressure ;
    gSP_RSGlue.MaxPressure := stSP_ColdGlue.MaxPressure ;
    gSP_RSGlue.ManPressure := stSP_ColdGlue.ManPressure ;
    gSP_RSGlue.AutoOnSpeed := stSP_ColdGlue.AutoOnSpeed ;
  END_IF ;

(* Glue Off/On From HMI *)
	HGW_2StatePB_0.PB := EDGEPOS(Glue_PB);
	GlueText_Ind := HGW_2StatePB_0.Text_Ind;
	GlueColor_Ind := HGW_2StatePB_0.Color_Ind;
	Glue_On := HGW_2StatePB_0.State1;
	HGW_2StatePB_0();

(* Glue Manual/Auto From HMI *)
	HGW_2StatePB_1.PB := (EDGEPOS(GlueAuto_PB) OR (NOT Glue_Auto AND gA[9].Ind_InMotion));
	GlueAutoText_Ind := HGW_2StatePB_1.Text_Ind;
	GlueAutoColor_Ind := HGW_2StatePB_1.Color_Ind;
	Glue_Auto := HGW_2StatePB_1.State1;
	HGW_2StatePB_1();

(* Glue Auto Pressure Based On Machine Speed *)
	HGW_ScaleReal_0.Enable := Glue_Auto;
	HGW_ScaleReal_0.InputMin := 0.0;
	HGW_ScaleReal_0.InputMax := gr_rMaxLSFlexoP_mmin/3.2808;
	HGW_ScaleReal_0.InputRaw := gActualMachineSpeed_FPM;
	HGW_ScaleReal_0.ScaledMin := gSP_RSGlue.MinPressure ;
	HGW_ScaleReal_0.ScaledMax := gSP_RSGlue.MaxPressure ;
	PressureCmd := HGW_ScaleReal_0.ScaledOut;
	HGW_ScaleReal_0();

(* Glue Manual Pressure *)
	IF (NOT Glue_Auto) THEN
		PressureCmd := gSP_RSGlue.ManPressure;
	END_IF

(* Glue Pressure Command Limit 0-100% *)
	PressureCmd := LIMIT (0,PressureCmd, 100);

(* If Disabled, Reduce Pressure To Zero  *)
	IF (NOT Glue_On) THEN
		PressureCmd := 0;
	END_IF

(* Generate Analog Command To Seam Paste System Pressure *)
	HGW_ScaleReal_1.Enable := 1;
	HGW_ScaleReal_1.InputMin := 0.0;
	HGW_ScaleReal_1.InputMax := 100.0;
	HGW_ScaleReal_1.InputRaw := PressureCmd;
	HGW_ScaleReal_1.ScaledMin := 0.0;
	HGW_ScaleReal_1.ScaledMax := 32767.0;
  gQ_CMD_RS_GluePressure  := REAL_TO_INT(HGW_ScaleReal_1.ScaledOut);
	HGW_ScaleReal_1();

(* Glue Auto On *)
  IF ((gActualMachineSpeed_FPM>=gSP_RSGlue.AutoOnSpeed) AND gA[9].Ind_InMotion AND Glue_On AND gBagMachine_WebBreakOK AND NOT(g_bIndEStop) ) THEN
		GlueAuto_On := 1;
	ELSE
		GlueAuto_On := 0;
	END_IF

(* Glue Gun Clean Control *)
	HGW_Toggle_0(In := GlueClean_PB , Time := T#12ms);

(* Glue Gun Control *)
	IF ( (GlueAuto_On OR GluePurge_PB OR HGW_Toggle_0.Out) AND gBagMachine_WebBreakOK AND gI_SS_SeamGlueOnOff AND NOT(g_bIndEStop) ) THEN
		gQ_CR_RS_Glue := 1;
	ELSE
		gQ_CR_RS_Glue := bTest1;
	END_IF

(* Is 2nd Tube Selected *)
	IF (gSP_TubeSelect) THEN
		gQ_CR_ColdGlueSelect := 1;
	ELSE
		gQ_CR_ColdGlueSelect := bTest2;
	END_IF

END_PROGRAM
```

#### RS_GlueInit.st
```iecst
(********************************************************************
 * COPYRIGHT -- Microsoft
 ********************************************************************
 * Program: RS_Glue
 * File: RS_GlueInit.st
 * Author: dominique
 * Created: October 26, 2011
 ********************************************************************
 * Implementation of program ColdGlue
 ********************************************************************)

PROGRAM _INIT

(* Glue Off/On PB Colors *)
	HGW_2StatePB_0.BackColor_State0 := gBlue;
	HGW_2StatePB_0.ForeColor_State0 := gWhite;
	HGW_2StatePB_0.BackColor_State1 := gGreen;
	HGW_2StatePB_0.ForeColor_State1 := gBlack;

(* Glue Manual/Auto PB Colors *)
	HGW_2StatePB_1.BackColor_State0 := gYellow;
	HGW_2StatePB_1.ForeColor_State0 := gBlack;
	HGW_2StatePB_1.BackColor_State1 := gGreen;
	HGW_2StatePB_1.ForeColor_State1 := gBlack;

  bTest1 := 0 ;
  bTest2 := 0 ;

END_PROGRAM
```

### Program Logical/BagMachine_Section/RS_Glue_V0

#### RS_Glue.var
```iecst
(********************************************************************
 * COPYRIGHT -- Microsoft
 ********************************************************************
 * Program: RS_Glue
 * File: RS_Glue.var
 * Author: dominique
 * Created: October 26, 2011
 ********************************************************************
 * Local variables of program ColdGlue
 ********************************************************************)
VAR
	Glue_Auto         : BOOL;
	Glue_On           : BOOL;
	Glue_PB           : BOOL;
	GlueAuto_On       : BOOL;
	GlueAuto_PB       : BOOL;
	GlueAutoColor_Ind : UINT;
	GlueAutoText_Ind  : UINT;
	GlueColor_Ind     : UINT;
	GluePurge_PB      : BOOL;
	GlueText_Ind      : UINT;
  rGlueMinPress     : REAL ;
  rGlueMaxPress     : REAL ;
  bTest1            : BOOL ;
  bTest2            : BOOL ;

  stSP_ColdGlue : Glue ;
  stSP_HotGlue  : Glue ;
END_VAR
VAR RETAIN
	HGW_2StatePB_0 : HGW_2StatePB;
	HGW_2StatePB_1 : HGW_2StatePB;
  rRS_ColdGlueMinPress : REAL ;
  rRS_HotGlueMinPress  : REAL ;
END_VAR
VAR
	HGW_ScaleReal_0 : HGW_ScaleReal;
	HGW_ScaleReal_1 : HGW_ScaleReal;
	PressureCmd : REAL;
	GlueClean_PB : BOOL;
	HGW_Toggle_0 : HGW_Toggle;
END_VAR
```

#### RS_GlueCyclic.st
```iecst
(********************************************************************
 * COPYRIGHT -- Microsoft
 ********************************************************************
 * Program: RS_Glue
 * File: RS_GlueeCyclic.st
 * Author: dominique
 * Created: October 26, 2011
 ********************************************************************
 * Implementation of program ColdGlue
 ********************************************************************)

PROGRAM _CYCLIC
  // Limit operator setpoint
  gSP_ColdGlue.MinPressure := LIMIT (0,gSP_ColdGlue.MinPressure,99) ;
  gSP_ColdGlue.MaxPressure := LIMIT (0,gSP_ColdGlue.MaxPressure,100) ;

  // Type RS glue selection (Cold/Hot)
  gQ_CR_HotColdGlueSelect := gRecipeActive.bSelTypeRSGlue ;
  IF EDGEPOS(gRecipeActive.bSelTypeRSGlue) THEN
    rRS_ColdGlueMinPress := gSP_ColdGlue.MinPressure ;
    gSP_ColdGlue.MinPressure := rRS_HotGlueMinPress ;
  END_IF ;
  IF EDGENEG(gRecipeActive.bSelTypeRSGlue) THEN
    rRS_HotGlueMinPress := gSP_ColdGlue.MinPressure ;
    gSP_ColdGlue.MinPressure := rRS_ColdGlueMinPress ;
  END_IF ;

(* Glue Off/On From HMI *)
	HGW_2StatePB_0.PB := EDGEPOS(Glue_PB);
	GlueText_Ind := HGW_2StatePB_0.Text_Ind;
	GlueColor_Ind := HGW_2StatePB_0.Color_Ind;
	Glue_On := HGW_2StatePB_0.State1;
	HGW_2StatePB_0();

(* Glue Manual/Auto From HMI *)
	HGW_2StatePB_1.PB := (EDGEPOS(GlueAuto_PB) OR (NOT Glue_Auto AND gA[9].Ind_InMotion));
	GlueAutoText_Ind := HGW_2StatePB_1.Text_Ind;
	GlueAutoColor_Ind := HGW_2StatePB_1.Color_Ind;
	Glue_Auto := HGW_2StatePB_1.State1;
	HGW_2StatePB_1();

(* Glue Auto Pressure Based On Machine Speed *)
	HGW_ScaleReal_0.Enable := Glue_Auto;
	HGW_ScaleReal_0.InputMin := 0.0;
	HGW_ScaleReal_0.InputMax := 1000.0;
	HGW_ScaleReal_0.InputRaw := gActualMachineSpeed_FPM;
	HGW_ScaleReal_0.ScaledMin := gSP_ColdGlue.MinPressure ;
	HGW_ScaleReal_0.ScaledMax := gSP_ColdGlue.MaxPressure ;
	PressureCmd := HGW_ScaleReal_0.ScaledOut;
	HGW_ScaleReal_0();

(* Glue Manual Pressure *)
	IF (NOT Glue_Auto) THEN
		PressureCmd := gSP_ColdGlue.ManPressure;
	END_IF

(* Glue Pressure Command Limit 0-100% *)
	PressureCmd := LIMIT (0,PressureCmd, 100);

(* If Disabled, Reduce Pressure To Zero  *)
	IF (NOT Glue_On) THEN
		PressureCmd := 0;
	END_IF

(* Generate Analog Command To Seam Paste System Pressure *)
	HGW_ScaleReal_1.Enable := 1;
	HGW_ScaleReal_1.InputMin := 0.0;
	HGW_ScaleReal_1.InputMax := 100.0;
	HGW_ScaleReal_1.InputRaw := PressureCmd;
	HGW_ScaleReal_1.ScaledMin := 0.0;
	HGW_ScaleReal_1.ScaledMax := 32767.0;
	//gQ_CMD_ColdGluePressure := REAL_TO_INT(HGW_ScaleReal_1.ScaledOut);
  gQ_CMD_RS_GluePressure  := REAL_TO_INT(HGW_ScaleReal_1.ScaledOut);
	HGW_ScaleReal_1();

(* Glue Auto On *)
  IF ((gActualMachineSpeed_FPM>=gSP_ColdGlue.AutoOnSpeed) AND gA[9].Ind_InMotion AND Glue_On AND gBagMachine_WebBreakOK) THEN
		GlueAuto_On := 1;
	ELSE
		GlueAuto_On := 0;
	END_IF

(* Glue Gun Clean Control *)
	HGW_Toggle_0(In := GlueClean_PB , Time := T#12ms);

(* Glue Gun Control *)
	IF ((GlueAuto_On OR GluePurge_PB OR HGW_Toggle_0.Out) AND gBagMachine_WebBreakOK AND gI_SS_SeamGlueOnOff) THEN
		gQ_CR_RS_Glue := 1;
	ELSE
		gQ_CR_RS_Glue := bTest1;
	END_IF

(* Is 2nd Tube Selected *)
	IF (gSP_TubeSelect) THEN
		gQ_CR_ColdGlueSelect := 1;
	ELSE
		gQ_CR_ColdGlueSelect := bTest2;
	END_IF

END_PROGRAM
```

### Data object Logical/BagMachine_Section/Servo_Power_Supply/Axis0/A0_Init (Ax) - Servo Power Supply Initialization File

#### A0_Init.ax
```
InitParameter (Version=2.14.0, NcSwId=ACP10)
  ACP10AXIS_typ:
    dig_in:
      level:
        reference = ncACTIV_HI
        pos_hw_end = ncACTIV_HI
        neg_hw_end = ncACTIV_HI
        trigger1 = ncACTIV_HI
        trigger2 = ncACTIV_HI
    encoder_if:
      parameter:
        count_dir = ncSTANDARD
        scaling:
          load:
            units = 1000
            rev_motor = 1
    limit:
      parameter:
        v_pos = 10000.0
        v_neg = 10000.0
        a1_pos = 50000.0
        a2_pos = 50000.0
        a1_neg = 50000.0
        a2_neg = 50000.0
        t_jolt = 0.0
        t_in_pos = 0.0
        pos_sw_end = 2000000000
        neg_sw_end = -2000000000
        ds_warning = 500.0
        ds_stop = 1000.0
        a_stop = 1e+030
    controller:
      mode = ncPOSITION
      position:
        kv = 50.0
        tn = 0.0
        t_predict = 0.0008
        t_total = 0.0008
        p_max = 10000.0
        i_max = 0.0
      speed:
        kv = 2.0
        tn = 0.0
        t_filter = 0.0
        isq_filter1:
          type = ncOFF
          a0 = 0.0
          a1 = 0.0
          b0 = 0.0
          b1 = 0.0
          b2 = 0.0
          c0_par_id = 0
          c1_par_id = 0
        isq_filter2:
          type = ncOFF
          a0 = 0.0
          a1 = 0.0
          b0 = 0.0
          b1 = 0.0
          b2 = 0.0
          c0_par_id = 0
          c1_par_id = 0
        isq_filter3:
          type = ncOFF
          a0 = 0.0
          a1 = 0.0
          b0 = 0.0
          b1 = 0.0
          b2 = 0.0
          c0_par_id = 0
          c1_par_id = 0
      uf:
        type = ncLINEAR
        auto_config = ncMOTOR_PAR
        u0 = 0.0
        un = 0.0
        fn = 50.0
        k_f_slip = 0.0
      ff:
        torque_load = 0.0
        torque_pos = 0.0
        torque_neg = 0.0
        kv_torque = 0.0
        inertia = 0.0
        t_filter_a = 0.0
    move:
      stop:
        parameter[0]:
          decel_ramp = ncA_LIMIT
          controller = ncON
        parameter[1]:
          decel_ramp = ncA_LIMIT
          controller = ncON
        parameter[2]:
          decel_ramp = ncA_LIMIT
          controller = ncON
        parameter[3]:
          decel_ramp = ncA_LIMIT
          controller = ncON
        quickstop:
          decel_ramp = ncA_LIMIT
      homing:
        parameter:
          s = 0
          v_switch = 5000.0
          v_trigger = 500.0
          a = 50000.0
          mode = ncDIRECT
          edge_sw = ncPOSITIVE
          start_dir = ncPOSITIVE
          trigg_dir = ncPOSITIVE
          ref_pulse = ncOFF
          tr_s_block = 0.0
      basis:
        parameter:
          v_pos = 10000.0
          v_neg = 10000.0
          a1_pos = 50000.0
          a2_pos = 50000.0
          a1_neg = 50000.0
          a2_neg = 50000.0
    message:
      text:
        parameter:
          format = ncBREAK
          columns = 80
          data_modul = Error_Eng
```

- Data object Logical/BagMachine_Section/Servo_Power_Supply/Axis0/A0_Par (Apt) - Servo Power Supply Parameter File (no source held here)

### Program Logical/BagMachine_Section/Servo_Power_Supply/Axis0/A0_Basic (IEC) - Basic Servo

#### A0_BasicCyclic.st
```iecst
(********************************************************************
 * COPYRIGHT -- Microsoft
 ********************************************************************
 * Program: A0_Basic
 * File: A0_BasicCyclic.st
 * Author: pkiel
 * Created: July 17, 2011
 ********************************************************************
 * Implementation of program A0_Basic
 ********************************************************************)

PROGRAM _CYCLIC

	IF(gA[0].Ident <> 0)THEN

	(************************ READ DRIVE STATUS *************************)
	(* Access to the following bools:
	gA[x]_DriveStatus.Simulation			: If TRUE, simulation mode is active
	gA[x]_DriveStatus.NetworkInit			: If TRUE, the network is initialized
	gA[x]_DriveStatus.HomeSwitch			: If TRUE, the digital reference switch input is active
	gA[x]_DriveStatus.PosHWSwitch			: If TRUE, the positive hardware end switch is active
	gA[x]_DriveStatus.NegHWSwitch			: If TRUE, the negative hardware end switch is active
	gA[x]_DriveStatus.Trigger1				: If TRUE, the first trigger input is active
	gA[x]_DriveStatus.Trigger2				: If TRUE, the second trigger input is active
	gA[x]_DriveStatus.DriveEnable			: If TRUE, the enable input is active
	gA[x]_DriveStatus.ControllerReady		: If TRUE, the controller is ready to beturned on
	gA[x]_DriveStatus.ControllerStatus		: If TRUE, the controller is turned on (Same as MC_Power.Status)
	gA[x]_DriveStatus.AxisError				: If TRUE, at least one error has occurred (not acknowledged)
	gA[x]_DriveStatus.LagWarning			: If TRUE, the lag error has exceeded the limit value specified for a warning*)
		MC_BR_ReadDriveStatus_0.Enable := 1;
		MC_BR_ReadDriveStatus_0.Axis := gA[0].Ident;
		MC_BR_ReadDriveStatus_0.AdrDriveStatus := ADR (DriveStatus);
		MC_BR_ReadDriveStatus_0();
		gA[0].Ind_Simulation		:=	DriveStatus.Simulation;
		gA[0].Ind_NetworkInit		:=	DriveStatus.NetworkInit;
		gA[0].Input_Home			:=	DriveStatus.HomeSwitch;
		gA[0].Input_PosHW			:=	DriveStatus.PosHWSwitch;
		gA[0].Input_NegHW			:=	DriveStatus.NegHWSwitch;
		gA[0].Input_Trigger1		:=	DriveStatus.Trigger1;
		gA[0].Input_Trigger2		:=	DriveStatus.Trigger2;
		gA[0].Input_DriveEnable		:=	DriveStatus.DriveEnable;
		gA[0].Ind_ControllerReady	:=	DriveStatus.ControllerReady;
		gA[0].Ind_ControllerStatus	:=	DriveStatus.ControllerStatus;
		gA[0].Error					:=	DriveStatus.AxisError;
		gA[0].Ind_LagWarning		:=	DriveStatus.LagWarning;

			(************************ READ AXIS ERROR **********************)
		MC_ReadAxisError_0.Enable := gA[0].Ind_NetworkInit;
		MC_ReadAxisError_0.Axis := gA[0].Ident;
		MC_ReadAxisError_0.DataAddress := ADR(gA[0].ErrorText);
		MC_ReadAxisError_0.DataLength := SIZEOF(gA[0].ErrorText);
		MC_ReadAxisError_0.DataObjectName := 'Error_Eng';
		MC_ReadAxisError_0();
		IF(MC_ReadAxisError_0.Valid) THEN
			gA[0].ErrorID := MC_ReadAxisError_0.AxisErrorID;
			gA[0].ErrorCount := MC_ReadAxisError_0.AxisErrorCount;
		END_IF
		(* Auto Acknowledge Errors *)
		IF (gA[0].Cmd_Reset AND (gA[0].ErrorCount<>0) AND NOT AutoAck) THEN
			AutoAck:=1;
		ELSE
			AutoAck:=0;
		END_IF
		(*Axis Error Acknowledge*)
		IF (EDGEPOS(AutoAck) OR EDGEPOS(gA[0].ErrorAck)) THEN
			MC_ReadAxisError_0.Acknowledge := 1;
		ELSE;
			MC_ReadAxisError_0.Acknowledge :=0;
		END_IF

		(************************ RESET AXIS ERROR **********************)
		IF (gA[0].Cmd_Reset AND (gA[0].ErrorCount=0) AND gA[0].ErrorStop) THEN
			MC_Reset_0.Execute:=1;
			gA[0].Cmd_Reset:=0;
		END_IF
		IF (MC_Reset_0.Done) THEN
			MC_Reset_0.Execute:=0;
		END_IF
		MC_Reset_0.Axis:=gA[0].Ident;
		MC_Reset_0();

		(************************ READ AXIS STATUS *************************)
		MC_ReadStatus_0.Enable := gA[0].Ind_NetworkInit;
		MC_ReadStatus_0.Axis := gA[0].Ident;
		MC_ReadStatus_0();
		IF(MC_ReadStatus_0.Valid = TRUE)THEN
			gA[0].Ind_Enabled 			:= NOT (MC_ReadStatus_0.Disabled);
			gA[0].Ind_StandStill		:= MC_ReadStatus_0.StandStill;
			gA[0].Ind_Stopping			:= MC_ReadStatus_0.Stopping;
			gA[0].Ind_DiscreteMotion	:= MC_ReadStatus_0.DiscreteMotion;
			gA[0].Ind_ContinuousMotion	:= MC_ReadStatus_0.ContinuousMotion;
			gA[0].Ind_SynchronizedMotion:= MC_ReadStatus_0.SynchronizedMotion;
			gA[0].ErrorStop				:= MC_ReadStatus_0.Errorstop;
		END_IF

		(************************ ENABLE POWER SUPPLY **********************)
		MC_Power_0.Axis:=gA[0].Ident;
		IF (MC_Power_0.Error=0 AND NOT gA[0].ErrorStop) THEN
      MC_Power_0.Enable:= gQ_CR_MainPowerOn ;
		ELSE;
			MC_Power_0.Enable:=0;
		END_IF;
		MC_Power_0();

		IF (gA[0].Ind_Enabled AND NOT gA[0].ErrorStop AND gPowerUp_Complete) THEN
			gDriveSupply_Ready := 1;
		ELSE
			gDriveSupply_Ready :=0;
		END_IF

		(* Cyclic Read: Power Supply Current *)
		MC_BR_PowerMeter_0.Axis := gA[0].Ident;
        MC_BR_PowerMeter_0.IntervalTime:=60000;
        MC_BR_PowerMeter_0.Mode:=mcONLY_PSM;

		MC_BR_PowerMeter_0();

	END_IF

END_PROGRAM
```

- Program Logical/BagMachine_Section/Tearing/Axis4/A4_Automat (IEC) (no source held here)

### Program Logical/BagMachine_Section/Tearing/Axis4/A4_Basic

#### A4_BasicCyclic.st
```iecst
(********************************************************************
 * COPYRIGHT -- Microsoft
 ********************************************************************
 * Program: A4_Basic
 * File: A4_BasicCyclic.st
 * Author: pkiel
 * Created: July 13, 2011
 ********************************************************************
 * Implementation of program A4_Basic
 ********************************************************************)

PROGRAM _CYCLIC

	(* Theoretical Diameter = 4.7" *)
	(*gSP_A[1].Diameter := LIMIT (4.6,gSP_A[1].Diameter,4.8);*)
	(*gA[4].UnitsPerInch := gA[4].AxisPeriod/(gSP_A[1].Diameter*PI);*)
	gA[4].UnitsPerInch := gA[4].AxisPeriod/gRecipeActive.Repeat;
  gA[4].InchPerDeg := gA[4].UnitsPerDeg / gA[4].UnitsPerInch ;

	IF (gA[4].Ident<>0) THEN

	(************************ READ DRIVE STATUS *************************)
	(* Access to the following bools:
	gA[x]_DriveStatus.Simulation			: If TRUE, simulation mode is active
	gA[x]_DriveStatus.NetworkInit			: If TRUE, the network is initialized
	gA[x]_DriveStatus.HomeSwitch			: If TRUE, the digital reference switch input is active
	gA[x]_DriveStatus.PosHWSwitch			: If TRUE, the positive hardware end switch is active
	gA[x]_DriveStatus.NegHWSwitch			: If TRUE, the negative hardware end switch is active
	gA[x]_DriveStatus.Trigger1				: If TRUE, the first trigger input is active
	gA[x]_DriveStatus.Trigger2				: If TRUE, the second trigger input is active
	gA[x]_DriveStatus.DriveEnable			: If TRUE, the enable input is active
	gA[x]_DriveStatus.ControllerReady		: If TRUE, the controller is ready to beturned on
	gA[x]_DriveStatus.ControllerStatus		: If TRUE, the controller is turned on (Same as MC_Power.Status)
	gA[x]_DriveStatus.AxisError				: If TRUE, at least one error has occurred (not acknowledged)
	gA[x]_DriveStatus.LagWarning			: If TRUE, the lag error has exceeded the limit value specified for a warning*)
		MC_BR_ReadDriveStatus_0.Enable := 1;
		MC_BR_ReadDriveStatus_0.Axis := gA[4].Ident;
		MC_BR_ReadDriveStatus_0.AdrDriveStatus := ADR (DriveStatus);
		MC_BR_ReadDriveStatus_0();
		gA[4].Ind_Simulation		:=	DriveStatus.Simulation;
		gA[4].Ind_NetworkInit		:=	DriveStatus.NetworkInit;
		gA[4].Input_Home			:=	DriveStatus.HomeSwitch;
		gA[4].Input_PosHW			:=	DriveStatus.PosHWSwitch;
		gA[4].Input_NegHW			:=	DriveStatus.NegHWSwitch;
		gA[4].Input_Trigger1		:=	DriveStatus.Trigger1;
		gA[4].Input_Trigger2		:=	DriveStatus.Trigger2;
		gA[4].Input_DriveEnable		:=	DriveStatus.DriveEnable;
		gA[4].Ind_ControllerReady	:=	DriveStatus.ControllerReady;
		gA[4].Ind_ControllerStatus	:=	DriveStatus.ControllerStatus;
		gA[4].Error					:=	DriveStatus.AxisError;
		gA[4].Ind_LagWarning		:=	DriveStatus.LagWarning;

	(************************ READ AXIS ERROR **********************)
		MC_ReadAxisError_0.Enable := gA[4].Ind_NetworkInit;
		MC_ReadAxisError_0.Axis := gA[4].Ident;
		MC_ReadAxisError_0.DataAddress := ADR(gA[4].ErrorText);
		MC_ReadAxisError_0.DataLength := SIZEOF(gA[4].ErrorText);
		MC_ReadAxisError_0.DataObjectName := 'Error_Eng';
		MC_ReadAxisError_0();
		IF(MC_ReadAxisError_0.Valid) THEN
			gA[4].ErrorID := MC_ReadAxisError_0.AxisErrorID;
			gA[4].ErrorCount := MC_ReadAxisError_0.AxisErrorCount;
		END_IF
	(* Auto Acknowledge Errors *)
		IF (gA[4].Cmd_Reset AND (gA[4].ErrorCount<>0) AND NOT AutoAck) THEN
			AutoAck:=1;
		ELSE
			AutoAck:=0;
		END_IF
	(*Axis Error Acknowledge*)
		IF (EDGEPOS(AutoAck) OR EDGEPOS(gA[4].ErrorAck)) THEN
			MC_ReadAxisError_0.Acknowledge := 1;
		ELSE;
			MC_ReadAxisError_0.Acknowledge :=0;
		END_IF

	(************************ RESET AXIS ERROR **********************)
		IF (gA[4].Cmd_Reset AND (gA[4].ErrorCount=0) AND gA[4].ErrorStop) THEN
			MC_Reset_0.Execute:=1;
		END_IF
		IF (MC_Reset_0.Done) THEN
			MC_Reset_0.Execute:=0;
			gA[4].Cmd_Reset:=0;
			ResetError := 0;
		END_IF
		IF (MC_Reset_0.Error) THEN
			MC_Reset_0.Execute:=0;
			gA[4].Cmd_Reset:=0;
			ResetError := 1;
		END_IF
		MC_Reset_0.Axis:=gA[4].Ident;
		MC_Reset_0();

	(************************ READ AXIS STATUS *************************)
		MC_ReadStatus_0.Enable := gA[4].Ind_NetworkInit;
		MC_ReadStatus_0.Axis := gA[4].Ident;
		MC_ReadStatus_0();
		IF(MC_ReadStatus_0.Valid = TRUE)THEN
			gA[4].Ind_Enabled 			     := NOT (MC_ReadStatus_0.Disabled);
			gA[4].Ind_StandStill		     := MC_ReadStatus_0.StandStill;
			gA[4].Ind_Stopping		    	 := MC_ReadStatus_0.Stopping;
			gA[4].Ind_DiscreteMotion	   := MC_ReadStatus_0.DiscreteMotion;
			gA[4].Ind_ContinuousMotion	 := MC_ReadStatus_0.ContinuousMotion;
			gA[4].Ind_SynchronizedMotion := MC_ReadStatus_0.SynchronizedMotion;
			gA[4].ErrorStop := MC_ReadStatus_0.Errorstop;
		END_IF
    IF NOT(gA[4].Ind_Enabled) THEN
      gA[4].bSynchroReq := 1 ;
    END_IF
    IF EDGEPOS(gA[4].Ind_bSynchroOK) THEN
      gA[4].bSynchroReq := 0 ;
    END_IF

	(******************** INIT POSITION MODULUS  *********************)
    IF (g_rNumbPliers <> 0.0) THEN
      IF ( gA[4].Ind_StandStill     OR
           NOT(gA[4].Ind_Enabled) ) AND
         g_bChangeModTearingReq     THEN
        bChangeModReq := 1 ;
        uiInitModPos0_ErrorID := 0 ;
      END_IF
      MC_BR_InitModPos_0.Execute:= (InitModPosition OR bChangeModReq) ;
  		MC_BR_InitModPos_0.Axis:= gA[4].Ident;
  		MC_BR_InitModPos_0.Period:= REAL_TO_UDINT(gA[4].AxisPeriod * 4.0/g_rNumbPliers);
  		MC_BR_InitModPos_0.Factor:=1;
  		InitModPos_Done:=MC_BR_InitModPos_0.Done;
    END_IF
    IF MC_BR_InitModPos_0.Done THEN
      g_bChangeModTearingReq := 0 ;
      bChangeModReq          := 0 ;
    ELSIF MC_BR_InitModPos_0.Error THEN
      bChangeModReq := 0 ;
      uiInitModPos0_ErrorID := MC_BR_InitModPos_0.ErrorID ;
    END_IF
		MC_BR_InitModPos_0();

	(******************** INIT ENDLESS POSITION *********************)
		MC_BR_InitEndlessPosition_0.Execute:= InitModPos_Done;
		MC_BR_InitEndlessPosition_0.Axis:= gA[4].Ident;
		MC_BR_InitEndlessPosition_0.DataAddress:= ADR(gEndPosData[4]);
		IF (MC_BR_InitEndlessPosition_0.Done) THEN
			InitModPosition:=0;
			InitEndlessPosition:=0;
			HomeRestore:=1;
		END_IF
		MC_BR_InitEndlessPosition_0();

	(************************ HOME AXIS FIRST POWER UP **********************)
		IF (HomeRestore AND NOT gA4_FirstHomed) THEN
			MC_Home_0.Execute:=1;
		END_IF
		MC_Home_0.Axis:=gA[4].Ident;
		MC_Home_0.Position:=0;
		MC_Home_0.HomingMode:=mcHOME_DIRECT;
		IF (MC_Home_0.Done) THEN
			MC_Home_0.Execute:=0;
			gA4_FirstHomed:=1;
		END_IF
		MC_Home_0();

  (************************ HOME AXIS **********************)
    IF (gA4_FirstHomed) THEN
      MC_Home_1.Execute:=HomeRestore;
    END_IF
    MC_Home_1.Axis:=gA[4].Ident;
    MC_Home_1.Position:=0;
    MC_Home_1.HomingMode:=mcHOME_RESTORE_POS;
    IF (MC_Home_1.Done) THEN
      gA[4].Ind_Homed:=1;
      HomeRestore:=0;
    END_IF
    MC_Home_1();

  (************************ HOME AXIS **********************)
    IF ( gA[4].Ind_StandStill        OR
         NOT(gA[4].Ind_Enabled) )    AND
       ( g_bNumPliersChange4to2[1]   OR
         g_bNumPliersChange2to4[1] ) THEN
      MC_Home_2.Execute := 1 ;
      IF g_bNumPliersChange4to2[1] THEN
        rTemp_[2] := (gA[4].PositionDeg + 180.0) * gA[9].UnitsPerDeg ;
      ELSE
        rTemp_[2] := (gA[4].PositionDeg - 180.0) * gA[9].UnitsPerDeg ;
      END_IF
      rRedefPosTear := H_FC_Modulus (IN_rMod:=360*gA[4].rRSynNum/gA[4].rRSynDen,IN_rVar:=rTemp_[2]) ;
    END_IF
    MC_Home_2.Axis       := gA[4].Ident;
    MC_Home_2.Position   := rRedefPosTear ;
    MC_Home_2.HomingMode := mcHOME_DIRECT;
    IF (MC_Home_2.Done) THEN
      g_bNumPliersChange4to2[1] := 0 ;
      g_bNumPliersChange2to4[1] := 0 ;
      MC_Home_2.Execute := 0 ;
    END_IF
    IF MC_Home_2.Error THEN
      MC_Home_2.Execute := 0 ;
    END_IF
    MC_Home_2();

	(******************** READ ACTUAL POSITION *********************)
		MC_ReadActualPosition_0.Enable:= gA[4].Ind_NetworkInit;
		MC_ReadActualPosition_0.Axis:= gA[4].Ident;
		MC_ReadActualPosition_0();
		IF(MC_ReadActualPosition_0.Valid = TRUE)THEN
			gA[4].PositionCount := MC_ReadActualPosition_0.Position;
			gA[4].PositionInch := gA[4].PositionCount/gA[4].UnitsPerInch;
			gA[4].PositionDeg := gA[4].PositionCount/gA[4].UnitsPerDeg;
		END_IF

  //******************** READ SET POINT POSITION *********************
    // Slave side  : ParID 428 SGEN_S_SET : CTRL Position controller: Input set position
    // Master side : ParID 412 S_SET_VAX1 : 412: VAX: Position

    // Slave side
    MC_BR_CyclicRead_0.Axis        := gA[4].Ident ;
    MC_BR_CyclicRead_0.Enable      := gA[4].Ind_NetworkInit;
    MC_BR_CyclicRead_0.ParID       := 428 ;
    MC_BR_CyclicRead_0.DataAddress := ADR(iiSP_SlPos_U);
    MC_BR_CyclicRead_0.DataType    := ncPAR_TYP_DINT ;
    // Master side
    MC_BR_CyclicRead_1.Axis        := gA[9].Ident ;
    MC_BR_CyclicRead_1.Enable      := gA[4].Ind_NetworkInit;
    MC_BR_CyclicRead_1.ParID       := 412 ;
    MC_BR_CyclicRead_1.DataAddress := ADR(iiSP_MaPos_U);
    MC_BR_CyclicRead_1.DataType    := ncPAR_TYP_DINT ;

    IF MC_BR_CyclicRead_0.Valid THEN
      rSP_SlPos_Deg := iiSP_SlPos_U/gA[4].UnitsPerDeg ;
    ELSIF MC_BR_CyclicRead_0.Error THEN
      MC_BR_CyclicRead_0.Enable := 0 ;
    END_IF
    IF MC_BR_CyclicRead_1.Valid THEN
      rSP_MaPos_Deg := iiSP_MaPos_U/gA[9].UnitsPerDeg ;
    ELSIF MC_BR_CyclicRead_1.Error THEN
      MC_BR_CyclicRead_1.Enable := 0 ;
    END_IF
    MC_BR_CyclicRead_0();
    MC_BR_CyclicRead_1();

  //******************** READ ACTUAL OFFSET *********************
  IF gA[4].rRSynDen > 0.0 THEN
    rTempActPhasDeg := rSP_SlPos_Deg
                       - gA[4].rRSynNum / gA[4].rRSynDen
                       * rSP_MaPos_Deg;
    gA[4].rActPhasDeg := H_FC_Modulus (
                              IN_rMod := 360 * gA[4].rRSynNum / gA[4].rRSynDen ,
                              IN_rVar := rTempActPhasDeg
                                      ) ;
  END_IF

	(******************** READ ACTUAL VELOCITY *********************)
		IF(MC_ReadActualVelocity_0.Error=TRUE) THEN
			MC_ReadActualVelocity_0.Enable:= 0;
		ELSE
			MC_ReadActualVelocity_0.Enable:= 1;
		END_IF
		MC_ReadActualVelocity_0.Axis:= gA[4].Ident;
		MC_ReadActualVelocity_0();
		IF(MC_ReadActualVelocity_0.Valid = TRUE)THEN
      //gA[4].ActualVelocity := MC_ReadActualVelocity_0.Velocity*60/gA[4].SP_MotorPPR;
      gA[4].ActualVelocity := MC_ReadActualVelocity_0.Velocity*60/gA[4].AxisPeriod ; // D.M. 03/08/2011 BrownPaper_14542  Need speed of the axis and not of the shaft of the motor
			IF ABS(gA[4].ActualVelocity>1) THEN // D.M. 03/08/2011 BrownPaper_14542 Add ABS because in case negative velocity Ind_InMotion = 0 instead of 1
				gA[4].Ind_InMotion:=1;
			ELSE
				gA[4].Ind_InMotion:=0;
			END_IF
		END_IF

	(******************** READ ACTUAL TORQUE *********************)
		IF(MC_ReadActualTorque_0.Error=TRUE) THEN
			MC_ReadActualTorque_0.Enable:= 0;
		ELSE
			MC_ReadActualTorque_0.Enable:= 1;
		END_IF
		MC_ReadActualTorque_0.Axis:= gA[4].Ident;
		MC_ReadActualTorque_0();
		IF(MC_ReadActualTorque_0.Valid = TRUE)THEN
			gA[4].ActualTorque := MC_ReadActualTorque_0.Torque;
		END_IF

	(************************ ENABLE AXIS **********************)
		MC_Power_0.Axis:=gA[4].Ident;
		IF (MC_Power_0.Error=0) THEN
			MC_Power_0.Enable:=gA[4].Cmd_Enable;
		ELSE;
			MC_Power_0.Enable:=0;
		END_IF;
		MC_Power_0();

	(************************ AXIS VELOCITY MOVE **********************)
		MC_MoveVelocity_0.Axis:=gA[4].Ident;
		MC_MoveVelocity_0.Velocity:=gA[4].SP_Velocity*gA[4].AxisPeriod/60;
		MC_MoveVelocity_0.Acceleration:=gA[4].SP_Accel;
		MC_MoveVelocity_0.Deceleration:=gA[4].SP_Decel;
		MC_MoveVelocity_0.Direction:=mcPOSITIVE_DIR;
		IF ((EDGEPOS(gA[4].Cmd_ContinuousMotion)) OR (EDGEPOS(gA[4].Cmd_ContinuousMotionUpdate))) THEN
			MC_MoveVelocity_0.Execute:=1;
		ELSE
			MC_MoveVelocity_0.Execute:=0;
		END_IF;
		MC_MoveVelocity_0();

  //************************ AXIS OVERRIDE **********************
    MC_SetOverride_0.Axis      := gA[4].Ident ;
    MC_SetOverride_0.Enable    := gA[4].Cmd_Override ;
    MC_SetOverride_0.VelFactor := gA[4].rSP_OverrideV ;
    MC_SetOverride_0.AccFactor := gA[4].rSP_OverrideA ;
    IF (MC_SetOverride_0.Enabled) OR
       (MC_SetOverride_0.Error)   THEN
      gA[4].Cmd_Override := 0 ;
    END_IF
    MC_SetOverride_0();

	(************************ AXIS STOP **********************)
		MC_Stop_0.Axis:=gA[4].Ident;
		IF (gA[4].Ind_ContinuousMotion AND (NOT gA[4].Cmd_ContinuousMotion) AND gAlarmsOK) THEN
			MC_Stop_0.Deceleration:=gA[4].SP_Decel;
			MC_Stop_0.Execute:=1;
		END_IF;
		IF (MC_Stop_0.Done OR MC_Stop_0.CommandAborted OR MC_Stop_0.Error) THEN
			MC_Stop_0.Execute:=0;
		END_IF;
		MC_Stop_0();

  (************************  ESTOP **********************)
    MC_Stop_1.Axis:=gA[4].Ident;
    IF EDGEPOS(g_bIndEStopStandstill) THEN
      MC_Stop_1.Deceleration:=gA[4].SP_EStopDecel;
      MC_Stop_1.Execute:=1;
    END_IF;
    IF (MC_Stop_1.Done OR MC_Stop_1.CommandAborted OR MC_Stop_1.Error) THEN
      MC_Stop_1.Execute:=0;
      gA[4].Cmd_EStopDisable := 1 ;
    END_IF;
    IF NOT(g_bIndEStopStandstill) THEN
      gA[4].Cmd_EStopDisable := 0 ;
    END_IF;
    MC_Stop_1();

    //************************ AXIS PHASE CONTROL (Inches) First Step **********************
    IF EDGEPOS(gA[4].Cmd_PhaseOffset) THEN
      rSP_PhaseOffset := gA[4].SP_PhaseOffset ;
    END_IF;

    (************************ SHIFTING PERF CONTROL **********************)
    IF g_bCmdShiftA[4] THEN
      //rSP_ShiftTearing := g_iPerfShiftPos * gr_rIncrShiftPerf_mm/25.4 * gA[4].rRSynNum/gA[4].rRSynDen ;  // D.M. RS26_Pyrollpack_14661 CAUTION !!! Phasing acts on the master side and not slave side, replaced by the code below
      rSP_ShiftTearing := g_iPerfShiftPos * gr_rIncrShiftPerf_mm/25.4 ;
      g_iCountPerfShift[2] := g_iCountPerfShift[2] - 1 ;
      gA[4].Cmd_PhaseOffset := 1 ;
      g_bCmdShiftA[4] := 0 ;
    END_IF

    (************************ AXIS PHASE CONTROL (Inches)  Next Step **********************)
    MC_BR_Phasing_0.Slave:=gA[4].Ident;
    IF gA[4].Ind_SynchronizedMotion AND NOT(gstCycA[4].CycManTimSet.bSCyc) AND st_TON_0.Q THEN
      MC_BR_Phasing_0.Enable:=1;
    ELSE
      MC_BR_Phasing_0.Enable:=0;
    END_IF
    IF gA[4].Cmd_PhaseOffset                AND
       ( EDGENEG(gA[4].Ind_bInContactZone)  OR
         gRecipeActive.bSelEnvBProd )       AND
       ( EDGENEG(gA[12].Ind_bInContactZone) OR
         NOT(gRecipeActive.bSelEnvBProd) )  AND
       NOT(gstCycA[4].CycManTimSet.bSCyc)   THEN
      MC_BR_Phasing_0.InitData := 1 ;
      gA[4].Cmd_PhaseOffset := 0 ;
      rSP_PhaseOffsetVal := rSP_PhaseOffset + rSP_ShiftTearing ;
      // Calculation new phase Tearing/Master
      rTemp_[0] := (rSP_PhaseOffsetVal)/gA[4].InchPerDeg ;
      rTemp_[1] := gRecipeActive.rTearing_PhasMasterDeg + rTemp_[0]*gA[4].rRSynNum/gA[4].rRSynDen ;
      gRecipeActive.rTearing_PhasMasterDeg := H_FC_Modulus (IN_rMod := 360*gA[4].rRSynNum/gA[4].rRSynDen, IN_rVar := rTemp_[1]) ;
      rSP_ShiftTearing := 0.0 ;
      rSP_PhaseOffset := 0.0 ;
      iTest_[0] := iTest_[0] + 1 ;
      iIndx := REAL_TO_INT(H_FC_Modulus(IN_rMod:=9,IN_rVar:=iTest_[0])) ;
      rTest_[iIndx] := rTemp_[0] ;
    ELSE
      MC_BR_Phasing_0.InitData:=0;
    END_IF
    MC_BR_Phasing_0.Shift               := rSP_PhaseOffsetVal*gA[9].UnitsPerInch;
    MC_BR_Phasing_0.Velocity            := 6*gA[4].AxisPeriod/60;
    MC_BR_Phasing_0.Acceleration        := gA[4].SP_Decel;
    MC_BR_Phasing_0.ApplicationDistance := 0.4*gA[9].AxisPeriod * gA[4].rRSynNum/gA[4].rRSynDen;
    MC_BR_Phasing_0.ApplicationMode     := mcMASTER_DISTANCE_BASED;
    MC_BR_Phasing_0.ShiftMode           := mcRELATIVE;
    MC_BR_Phasing_0();

    (************************ AXIS PHASE CONTROL (Inches) TIMING SETTING **********************)
    IF gstCycA[4].CycManTimSet.bSCyc THEN
      IF gA[4].Cmd_ManuTimSetPlus THEN
        rAxisTimSet_SP_Vel := gr_rAxisTimSet_SP_Vel*gA[9].AxisPeriod/60 / (gA[4].rRSynNum/gA[4].rRSynDen) ;
      ELSE
        rAxisTimSet_SP_Vel := - gr_rAxisTimSet_SP_Vel*gA[9].AxisPeriod/60 / (gA[4].rRSynNum/gA[4].rRSynDen) ;
      END_IF
        rAxisTimSet_SP_Acc := gr_rAxisTimSet_SP_Acc*gA[9].AxisPeriod/60/60 / (gA[4].rRSynNum/gA[4].rRSynDen) ;
    END_IF

    MC_BR_Phasing_1.Slave                  := gA[4].Ident;
    MC_BR_Phasing_1.Enable                 := gstCycA[4].CycManTimSet.bCyc ;
    MC_BR_Phasing_1.InitData               := gstCycA[4].CycManTimSet.bSCyc ;
    MC_BR_Phasing_1.PerformVelocityControl := gstCycA[4].CycManTimSet.CmdMov ;
    MC_BR_Phasing_1.Velocity               := rAxisTimSet_SP_Vel ;
    MC_BR_Phasing_1.Acceleration           := rAxisTimSet_SP_Acc ;
    MC_BR_Phasing_1.ApplicationMode        := mcVELOCITY_CONTROL ;
    MC_BR_Phasing_1();
    st_TON_0(IN:=NOT(MC_BR_Phasing_1.Enable),PT:=T#100ms) ;

    IF NOT(gstCycA[4].CycManTimSet.CmdMov) AND
       MC_BR_Phasing_1.ShiftAttained       OR
       NOT(gstCycA[4].CycManTimSet.bCyc)   OR
       MC_BR_Phasing_1.Error               AND
       1                                   THEN
      gstCycA[4].CycManTimSet.CmdStop := 0 ;
    END_IF
	END_IF

END_PROGRAM
```

### Program Logical/BagMachine_Section/Tearing/Axis4/A4_Control

#### A4_ControlCyclic.ld
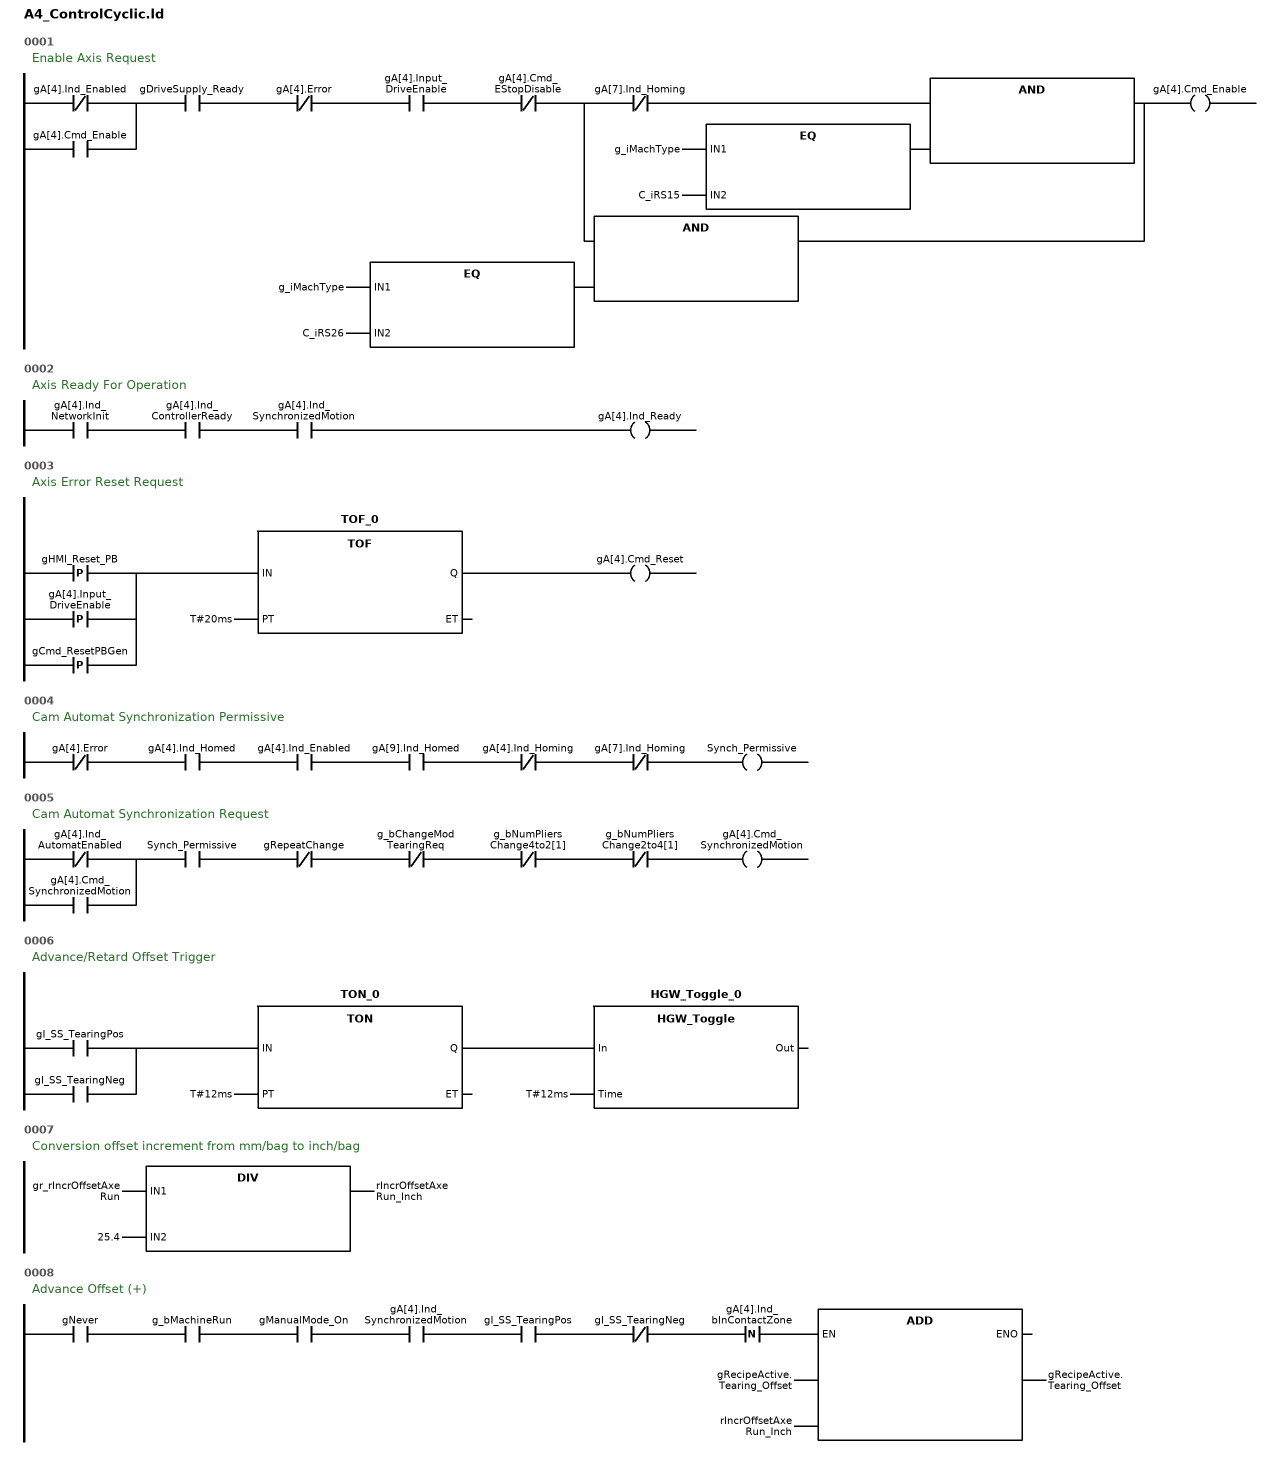
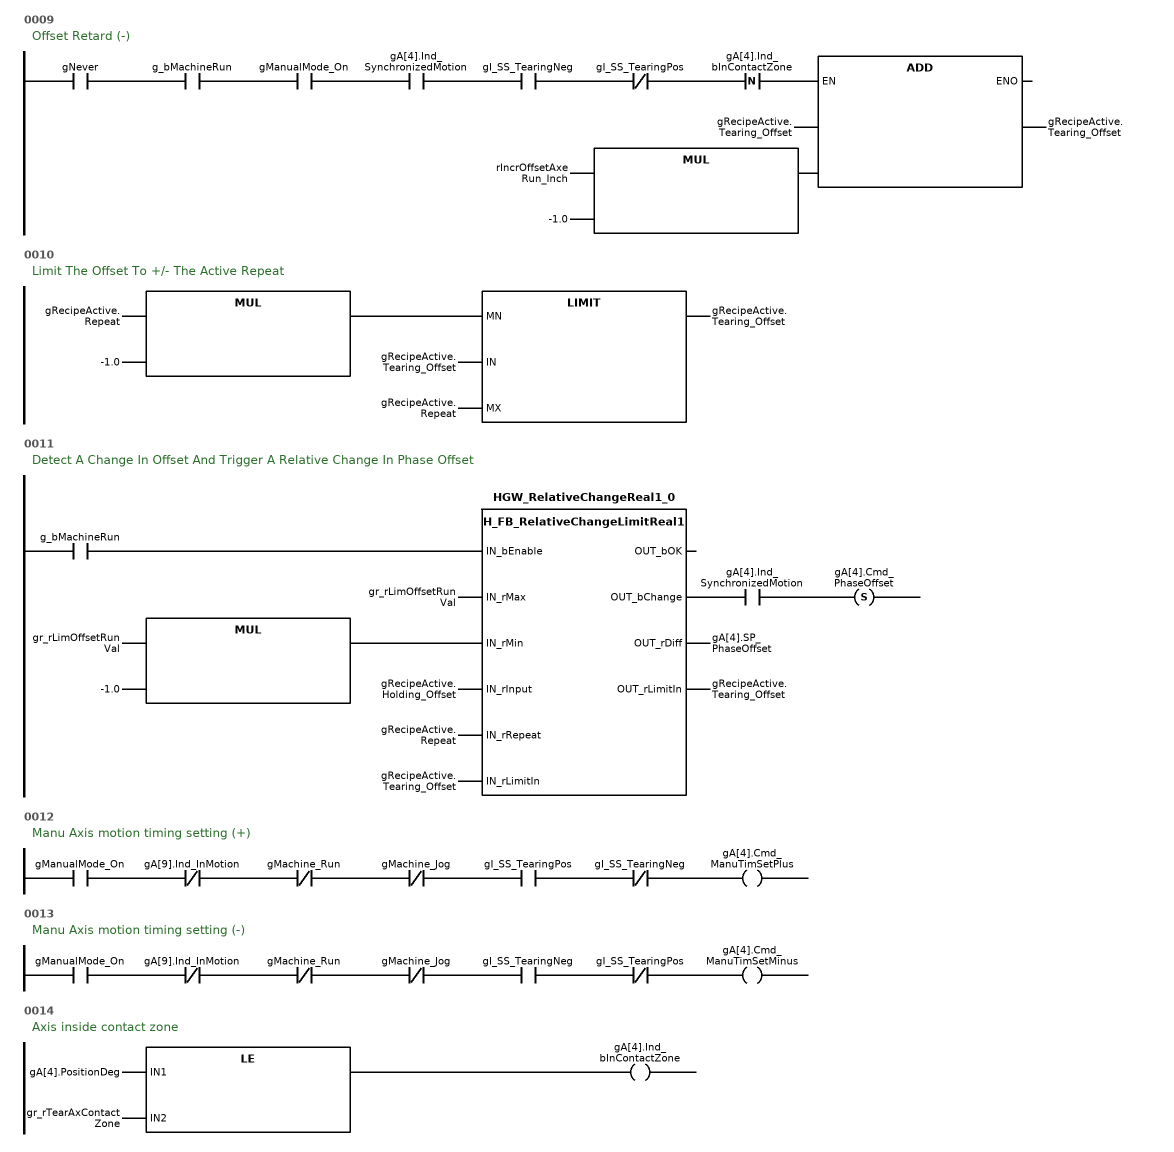
Ladder, written as Structured Text:
```iecst
(********************************************************************
 * COPYRIGHT -- Microsoft
 ********************************************************************
 * Program: A4_Control
 * File: A4_ControlCyclic.ld
 * Author: pkiel
 * Created: July 13, 2011
 ********************************************************************
 * Implementation of program A4_Control
 ********************************************************************)

PROGRAM _CYCLIC
VAR
    _p1 : BOOL;
    _e2 : R_TRIG;
    _e3 : R_TRIG;
    _e4 : R_TRIG;
    _e5 : F_TRIG;
    _e6 : F_TRIG;
END_VAR
(* Network 1: Enable Axis Request *)
_p1 := (NOT gA[4].Ind_Enabled OR gA[4].Cmd_Enable) AND gDriveSupply_Ready AND NOT gA[4].Error AND gA[4].Input_DriveEnable AND NOT gA[4].Cmd_EStopDisable;
gA[4].Cmd_Enable := _p1 AND ((NOT gA[7].Ind_Homing AND (g_iMachType = C_iRS15)) OR (g_iMachType = C_iRS26));

(* Network 2: Axis Ready For Operation *)
gA[4].Ind_Ready := gA[4].Ind_NetworkInit AND gA[4].Ind_ControllerReady AND gA[4].Ind_SynchronizedMotion;

(* Network 3: Axis Error Reset Request *)
_e2(CLK := gHMI_Reset_PB);
_e3(CLK := gA[4].Input_DriveEnable);
_e4(CLK := gCmd_ResetPBGen);
TOF_0(IN := _e2.Q OR _e3.Q OR _e4.Q, PT := T#20ms);
gA[4].Cmd_Reset := TOF_0.Q;

(* Network 4: Cam Automat Synchronization Permissive *)
Synch_Permissive := NOT gA[4].Error AND gA[4].Ind_Homed AND gA[4].Ind_Enabled AND gA[9].Ind_Homed AND NOT gA[4].Ind_Homing AND NOT gA[7].Ind_Homing;

(* Network 5: Cam Automat Synchronization Request *)
gA[4].Cmd_SynchronizedMotion := (NOT gA[4].Ind_AutomatEnabled OR gA[4].Cmd_SynchronizedMotion) AND Synch_Permissive AND NOT gRepeatChange AND NOT g_bChangeModTearingReq AND NOT g_bNumPliersChange4to2[1] AND NOT g_bNumPliersChange2to4[1];

(* Network 6: Advance/Retard Offset Trigger *)
TON_0(IN := gI_SS_TearingPos OR gI_SS_TearingNeg, PT := T#12ms);
HGW_Toggle_0(In := TON_0.Q, Time := T#12ms);

(* Network 7: Conversion offset increment from mm/bag to inch/bag *)
rIncrOffsetAxeRun_Inch := gr_rIncrOffsetAxeRun / 25.4;

(* Network 8: Advance Offset (+) *)
_e5(CLK := gA[4].Ind_bInContactZone);
IF gNever AND g_bMachineRun AND gManualMode_On AND gA[4].Ind_SynchronizedMotion AND gI_SS_TearingPos AND NOT gI_SS_TearingNeg AND _e5.Q THEN
    gRecipeActive.Tearing_Offset := gRecipeActive.Tearing_Offset + rIncrOffsetAxeRun_Inch;
END_IF;

(* Network 9: Offset Retard (-) *)
_e6(CLK := gA[4].Ind_bInContactZone);
IF gNever AND g_bMachineRun AND gManualMode_On AND gA[4].Ind_SynchronizedMotion AND gI_SS_TearingNeg AND NOT gI_SS_TearingPos AND _e6.Q THEN
    gRecipeActive.Tearing_Offset := gRecipeActive.Tearing_Offset + (rIncrOffsetAxeRun_Inch * -1.0);
END_IF;

(* Network 10: Limit The Offset To +/- The Active Repeat *)
gRecipeActive.Tearing_Offset := LIMIT(MN := gRecipeActive.Repeat * -1.0, IN := gRecipeActive.Tearing_Offset, MX := gRecipeActive.Repeat);

(* Network 11: Detect A Change In Offset And Trigger A Relative Change In Phase Offset *)
HGW_RelativeChangeReal1_0(IN_bEnable := g_bMachineRun, IN_rMax := gr_rLimOffsetRunVal, IN_rMin := gr_rLimOffsetRunVal * -1.0, IN_rInput := gRecipeActive.Holding_Offset, IN_rRepeat := gRecipeActive.Repeat, IN_rLimitIn := gRecipeActive.Tearing_Offset);
IF HGW_RelativeChangeReal1_0.OUT_bChange AND gA[4].Ind_SynchronizedMotion THEN
    gA[4].Cmd_PhaseOffset := TRUE;
END_IF;
gA[4].SP_PhaseOffset := HGW_RelativeChangeReal1_0.OUT_rDiff;
gRecipeActive.Tearing_Offset := HGW_RelativeChangeReal1_0.OUT_rLimitIn;

(* Network 12: Manu Axis motion timing setting (+) *)
gA[4].Cmd_ManuTimSetPlus := gManualMode_On AND NOT gA[9].Ind_InMotion AND NOT gMachine_Run AND NOT gMachine_Jog AND gI_SS_TearingPos AND NOT gI_SS_TearingNeg;

(* Network 13: Manu Axis motion timing setting (-) *)
gA[4].Cmd_ManuTimSetMinus := gManualMode_On AND NOT gA[9].Ind_InMotion AND NOT gMachine_Run AND NOT gMachine_Jog AND gI_SS_TearingNeg AND NOT gI_SS_TearingPos;

(* Network 14: Axis inside contact zone *)
gA[4].Ind_bInContactZone := gA[4].PositionDeg <= gr_rTearAxContactZone;
END_PROGRAM
```

- Program Logical/BagMachine_Section/Tearing/Axis4/A4_Cycle (IEC) (no source held here)

### Program Logical/BagMachine_Section/Tearing/Axis4/A4_Ref (IEC)

#### A4_RefCyclic.ld - Cyclic code
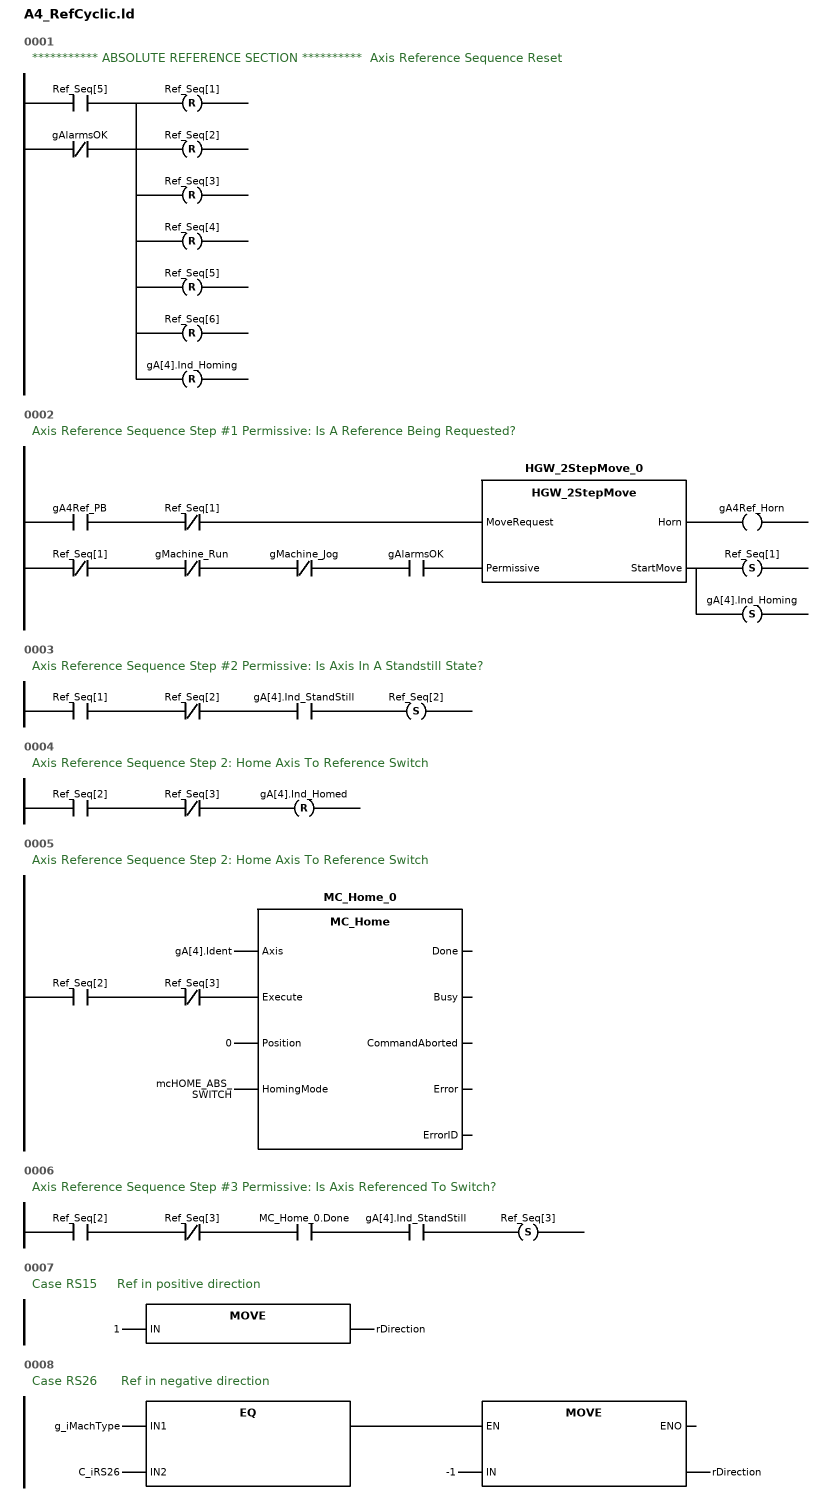
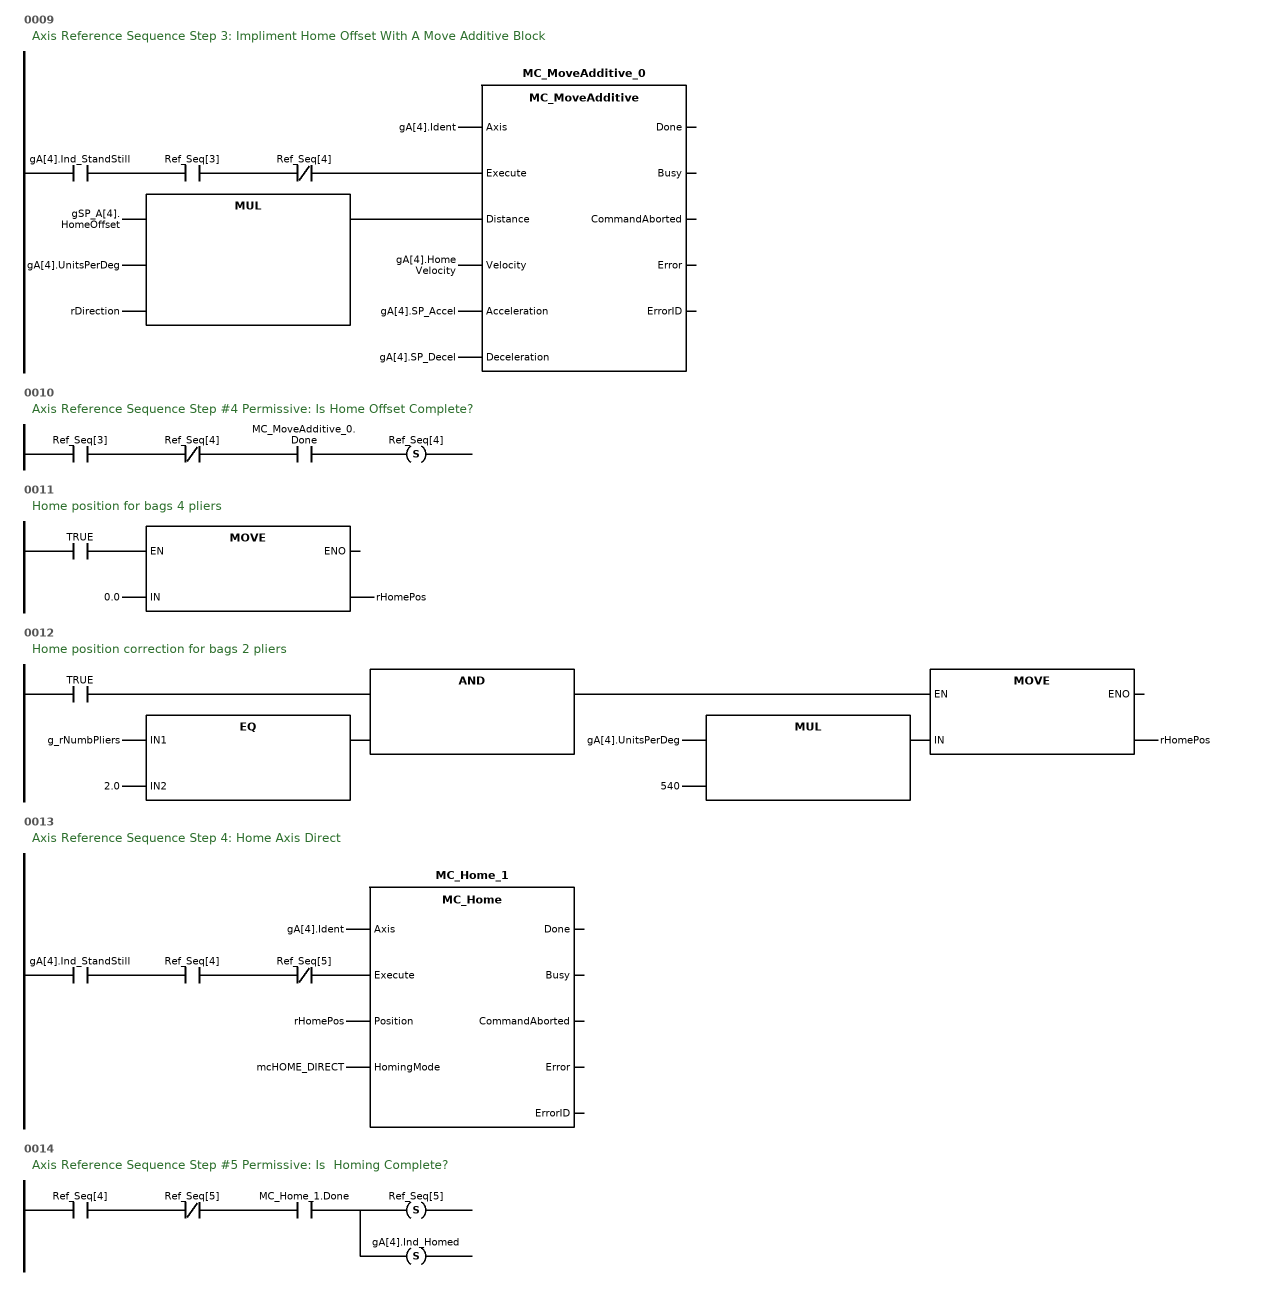
Ladder, written as Structured Text:
```iecst
(********************************************************************
 * COPYRIGHT -- Microsoft
 ********************************************************************
 * Program: A4_Ref
 * File: A4_RefCyclic.ld
 * Author: pkiel
 * Created: July 19, 2011
 ********************************************************************
 * Implementation of program A4_Ref
 ********************************************************************)

PROGRAM _CYCLIC
VAR
    _p1 : BOOL;
    _p2 : BOOL;
END_VAR
(* Network 1: *********** ABSOLUTE REFERENCE SECTION **********  Axis Reference Sequence Reset *)
_p1 := Ref_Seq[5];
IF Ref_Seq[5] OR NOT gAlarmsOK THEN Ref_Seq[1] := FALSE; END_IF;
IF _p1 OR NOT gAlarmsOK THEN
    Ref_Seq[2] := FALSE;
    Ref_Seq[3] := FALSE;
    Ref_Seq[4] := FALSE;
    Ref_Seq[5] := FALSE;
    Ref_Seq[6] := FALSE;
    gA[4].Ind_Homing := FALSE;
END_IF;

(* Network 2: Axis Reference Sequence Step #1 Permissive: Is A Reference Being Requested? *)
HGW_2StepMove_0(MoveRequest := gA4Ref_PB AND NOT Ref_Seq[1], Permissive := NOT Ref_Seq[1] AND NOT gMachine_Run AND NOT gMachine_Jog AND gAlarmsOK);
gA4Ref_Horn := HGW_2StepMove_0.Horn;
IF HGW_2StepMove_0.StartMove THEN
    Ref_Seq[1] := TRUE;
    gA[4].Ind_Homing := TRUE;
END_IF;

(* Network 3: Axis Reference Sequence Step #2 Permissive: Is Axis In A Standstill State? *)
IF Ref_Seq[1] AND NOT Ref_Seq[2] AND gA[4].Ind_StandStill THEN Ref_Seq[2] := TRUE; END_IF;

(* Network 4: Axis Reference Sequence Step 2: Home Axis To Reference Switch *)
IF Ref_Seq[2] AND NOT Ref_Seq[3] THEN gA[4].Ind_Homed := FALSE; END_IF;

(* Network 5: Axis Reference Sequence Step 2: Home Axis To Reference Switch *)
MC_Home_0(Axis := gA[4].Ident, Execute := Ref_Seq[2] AND NOT Ref_Seq[3], Position := 0, HomingMode := mcHOME_ABS_SWITCH);

(* Network 6: Axis Reference Sequence Step #3 Permissive: Is Axis Referenced To Switch? *)
IF Ref_Seq[2] AND NOT Ref_Seq[3] AND MC_Home_0.Done AND gA[4].Ind_StandStill THEN
    Ref_Seq[3] := TRUE;
END_IF;

(* Network 7: Case RS15     Ref in positive direction  *)
rDirection := 1;

(* Network 8: Case RS26      Ref in negative direction  *)
IF g_iMachType = C_iRS26 THEN rDirection := -1; END_IF;

(* Network 9: Axis Reference Sequence Step 3: Impliment Home Offset With A Move Additive Block *)
MC_MoveAdditive_0(Axis := gA[4].Ident, Execute := gA[4].Ind_StandStill AND Ref_Seq[3] AND NOT Ref_Seq[4], Distance := gSP_A[4].HomeOffset * gA[4].UnitsPerDeg * rDirection, Velocity := gA[4].HomeVelocity, Acceleration := gA[4].SP_Accel, Deceleration := gA[4].SP_Decel);

(* Network 10: Axis Reference Sequence Step #4 Permissive: Is Home Offset Complete? *)
IF Ref_Seq[3] AND NOT Ref_Seq[4] AND MC_MoveAdditive_0.Done THEN Ref_Seq[4] := TRUE; END_IF;

(* Network 11: Home position for bags 4 pliers  *)
rHomePos := 0.0;

(* Network 12: Home position correction for bags 2 pliers *)
IF g_rNumbPliers = 2.0 THEN rHomePos := gA[4].UnitsPerDeg * 540; END_IF;

(* Network 13: Axis Reference Sequence Step 4: Home Axis Direct *)
MC_Home_1(Axis := gA[4].Ident, Execute := gA[4].Ind_StandStill AND Ref_Seq[4] AND NOT Ref_Seq[5], Position := rHomePos, HomingMode := mcHOME_DIRECT);

(* Network 14: Axis Reference Sequence Step #5 Permissive: Is  Homing Complete? *)
_p2 := Ref_Seq[4] AND NOT Ref_Seq[5] AND MC_Home_1.Done;
IF Ref_Seq[4] AND NOT Ref_Seq[5] AND MC_Home_1.Done THEN Ref_Seq[5] := TRUE; END_IF;
IF _p2 THEN gA[4].Ind_Homed := TRUE; END_IF;
END_PROGRAM
```

#### A4_Ref.var - Local variables
```iecst
(********************************************************************
 * COPYRIGHT -- Microsoft
 ********************************************************************
 * Program: A4_Ref
 * File: A4_Ref.var
 * Author: pkiel
 * Created: July 19, 2011
 ********************************************************************
 * Local variables of program A4_Ref
 ********************************************************************)
VAR
	HGW_2StepMove_0 : HGW_2StepMove;
	MC_Home_0 : MC_Home;
	MC_Home_1 : MC_Home;
	MC_MoveAdditive_0 : MC_MoveAdditive;
	Ref_Seq : ARRAY[0..10] OF BOOL;

  rHomePos   : REAL ;
  rDirection : REAL ;
END_VAR
```

### Program Logical/BagMachine_Section/Unw_3W_Glue (IEC)

#### Unw_3W_GlueInit.st - Initialization code
```iecst
(********************************************************************
 * COPYRIGHT -- Microsoft
 ********************************************************************
 * Program: Unw_3W_Glue
 * File: Unw_3W_Glue.st
 * Author: dominique
 * Created: October 26, 2011
 ********************************************************************
 * Implementation of program Unw_3W_Glue
 ********************************************************************)

PROGRAM _INIT

(* Glue Off/On PB Colors *)
	HGW_2StatePB_0.BackColor_State0 := gBlue;
	HGW_2StatePB_0.ForeColor_State0 := gWhite;
	HGW_2StatePB_0.BackColor_State1 := gGreen;
	HGW_2StatePB_0.ForeColor_State1 := gBlack;

(* Glue Manual/Auto PB Colors *)
	HGW_2StatePB_1.BackColor_State0 := gYellow;
	HGW_2StatePB_1.ForeColor_State0 := gBlack;
	HGW_2StatePB_1.BackColor_State1 := gGreen;
	HGW_2StatePB_1.ForeColor_State1 := gBlack;

END_PROGRAM
```

#### Unw_3W_Glue.var - Local variables
```iecst
(********************************************************************
 * COPYRIGHT -- Microsoft
 ********************************************************************
 * Program: Unw_3W_Glue
 * File: Unw_3W_Glue.var
 * Author: dominique
 * Created: October 26, 2011
 ********************************************************************
 * Local variables of program Unw_3W_Glue
 ********************************************************************)
VAR
  iiSPDelayActGlue   : DINT ;
  tSPDelayActGlue    : TIME ;
  stTON_DelayActGlue : TON ;
  bImQ_CR_UNW_Glue   : BOOL ;

	Glue_Auto   : BOOL;
	Glue_On     : BOOL;
	Glue_PB     : BOOL;
	GlueAuto_On : BOOL;
	GlueAuto_PB : BOOL;
	GlueAutoColor_Ind : UINT;
	GlueAutoText_Ind  : UINT;
	GlueClean_PB  : BOOL;
	GlueColor_Ind : UINT;
	GluePurge_PB  : BOOL;
	GlueText_Ind  : UINT;
  rGlueMinPress : REAL ;
  rGlueMaxPress : REAL ;
  bQ_CR_3W_Glue2 : BOOL;
  bQ_CR_3W_GlueOn : BOOL;
  Glue3WAuto_On : BOOL;
  Glue3WAuto2_On : BOOL;

  HMI_rOtherRSGlueActPress : REAL ;
END_VAR
VAR RETAIN
	HGW_2StatePB_0 : HGW_2StatePB;
	HGW_2StatePB_1 : HGW_2StatePB;
  HMI_bSelHotColdRSGlue_PB : BOOL ;
  HMI_rSPDelayActGlue  : REAL ;
  stSP_ColdGlue : Glue ;
  stSP_HotGlue  : Glue ;
END_VAR

VAR
	HGW_ScaleReal_0 : HGW_ScaleReal;
	HGW_ScaleReal_1 : HGW_ScaleReal;
	HGW_Toggle_0 : HGW_Toggle;
	PressureCmd : REAL;
END_VAR
```

### Program Logical/BagMachine_Section/Unwinder (IEC)

#### UnwinderCyclic.st - Cyclic code
```iecst
(********************************************************************
 * COPYRIGHT -- .
 ********************************************************************
 * Program: Unwinder
 * File: UnwinderCyclic.st
 * Author: dominique
 * Created: August 10, 2011
 ********************************************************************
 * Implementation of program Unwinder
 ********************************************************************)

PROGRAM _CYCLIC

    // Brake WARNER on machine Pyrollpack_14661

 (* Terminal1 |  Brake Control (PID regulation)
    ----------|--------------------
       0      |      YES
    ----------|--------------------
       1      |      NO

    Terminal4 |  Lock Brake ( EStop )
    ----------|--------------------
       0      |      YES
    ----------|--------------------
       1      |      NO             *)

// ------------------------------------------------------------------------------------
// Brake management
    // Special case WARNER Brake on machine Pyrollpack_14661
    // Terminal1 on WARNER device (Control)
    bPIDRegul := g_bMainPower_On      AND
                 gA[9].Ind_InMotion   AND
                 1                    ;
    gQ_CR_UNW_PIDRegul := NOT(bPIDRegul) ;

    // Terminal4 on WARNER device (Lock)
    bLock := g_bMainPower_On     AND
             ( g_bIndStopFault   OR
               g_bIndStopFault ) AND
             1                   ;
    gQ_CR_UNW_Lock := NOT(bLock) AND
                      1          ;

// ------------------------------------------------------------------------------------
    // Enable regualtion on the customer's unwinder when master is in motion
    gQ_CR_UnwinRegEnable := gA[9].Ind_InMotion OR
                            bTest              ;

  // ------------------------------------------------------------------------------------
  // Regualtion on the HOLWEG unwinder when master is in motion
    // Input B on MEROBEL device
    bTemp := gI_SS_UNW_Brake    AND
             gA[9].Ind_InMotion ;
    gQ_CR_UNW_Brake := NOT(bTemp)                  AND
                       ( NOT(g_bIndStopFault)      AND
                         NOT(g_bIndEStop)          OR
                         NOT(gA[9].Ind_InMotion) ) AND
                       1                           ;

    // Input A on MEROBEL device
    gQ_CR_UNW_PIDRegul := gI_SS_UNW_Brake             AND
                          ( NOT(g_bIndStopFault)      AND
                            NOT(g_bIndEStop)          OR
                            NOT(gA[9].Ind_InMotion) ) AND
                          1                           ;

// ------------------------------------------------------------------------------------
// Forks management
    bForkUpReq   := gI_SS_UNW_ForkUp AND NOT(gI_SS_UNW_ForkDown) ;
    bForkDownReq := gI_SS_UNW_ForkDown AND NOT(gI_SS_UNW_ForkUp) ;
    bForkRequest := gI_SS_UNW_ForkUp OR gI_SS_UNW_ForkDown ;
    stTON_DelayActFork(IN:=bForkRequest, PT:=tDelayActFork) ;
    // Fork Up
    bImQ_CR_UNW_ForkUp := bForkUpReq         AND
                        stTON_DelayActFork.Q ;
    gQ_CR_UNW_ForkUp := bImQ_CR_UNW_ForkUp AND
                        NOT(g_bIndEStop)   ;
    // Fork Down
    bImQ_CR_UNW_ForkDown := bForkDownReq         AND
                            stTON_DelayActFork.Q ;
    gQ_CR_UNW_ForkDown := bImQ_CR_UNW_ForkDown AND
                          NOT(g_bIndEStop)     ;

    // Hydraulic Pump
    stTOF_ActHydroPump(IN:=bForkRequest, PT:=tTimActPump);
    bImQ_CR_UNW_HydroPump := stTOF_ActHydroPump.Q ;
    gQ_CR_UNW_HydroPump := bImQ_CR_UNW_HydroPump AND NOT(g_bIndEStop) ;

END_PROGRAM
```

#### UnwinderInit.st - Initialization code
```iecst
(********************************************************************
 * COPYRIGHT -- .
 ********************************************************************
 * Program: Unwinder
 * File: UnwinderInit.st
 * Author: dominique
 * Created: August 10, 2011
 ********************************************************************
 * Implementation of program Unwinder
 ********************************************************************)

PROGRAM _INIT

  tTimActPump   := T#1s ;
  tDelayActFork := T#0.5s ;

  bTest := 0 ;

END_PROGRAM
```

#### Unwinder.var - Local variables
```iecst
(********************************************************************
 * COPYRIGHT -- .
 ********************************************************************
 * Program: Unwinder
 * File: Unwinder.var
 * Author: dominique
 * Created: August 10, 2011
 ********************************************************************
 * Local variables of program Unwinder
 ********************************************************************)

VAR
  bImQ_CR_UNW_ForkUp    : BOOL ;
  bImQ_CR_UNW_ForkDown  : BOOL ;
  bImQ_CR_UNW_Brake     : BOOL ;
  bImQ_CR_UNW_HydroPump : BOOL ;
  stTOF_ActHydroPump    : TOF ;
  stTON_DelayActFork    : TON ;
  tTimActPump           : TIME := T#1s ;
  tDelayActFork         : TIME := T#0.5s ;
  bForkUpReq            : BOOL ;
  bForkDownReq          : BOOL ;
  bForkRequest          : BOOL ;

  bTemp     : BOOL ;
  bPIDRegul : BOOL ;
  bLock     : BOOL ;
  bTest     : BOOL := 0 ;
END_VAR

VAR CONSTANT
END_VAR
```

### Program Logical/BagMachine_Section/Vacuum (IEC)

#### VacuumInit.st - Initialization code
```iecst
(********************************************************************
 * COPYRIGHT -- Microsoft
 ********************************************************************
 * Program: Vacuum
 * File: VacuumInit.st
 * Author: pkiel
 * Created: July 19, 2011
 ********************************************************************
 * Implementation of program Vacuum
 ********************************************************************)

PROGRAM _INIT

(* Vacuum Off/On PB Colors *)
	HGW_2StatePB_0.BackColor_State0 := gBlue;
	HGW_2StatePB_0.ForeColor_State0 := gWhite;
	HGW_2StatePB_0.BackColor_State1 := gGreen;
	HGW_2StatePB_0.ForeColor_State1 := gBlack;

END_PROGRAM
```

#### Vacuum.var - Local variables
```iecst
(********************************************************************
 * COPYRIGHT -- Microsoft
 ********************************************************************
 * Program: Vacuum
 * File: Vacuum.var
 * Author: pkiel
 * Created: July 19, 2011
 ********************************************************************
 * Local variables of program Vacuum
 ********************************************************************)
VAR RETAIN
	HGW_2StatePB_0 : HGW_2StatePB;
END_VAR
VAR
	Vacuum_On : BOOL;
	Vacuum_PB : BOOL;
	VacuumColor_Ind : UINT;
	VacuumText_Ind : UINT;
END_VAR
```

### GenCycles.typ - Global data types
```iecst
TYPE
  MoveStat :
    (
    INACTIVE := 0 ,
    ACTIVE   := 1 ,
    FINISHED := 2 ,
    FAULT    := 3
    ) ;

  CycManTimSet : STRUCT
    bSCyc           : BOOL ;
    bFCyc           : BOOL ;
    bCyc            : BOOL ;
    bCycFail        : BOOL ;
    bModTest        : BOOL ;
    bTestOn         : BOOL ;
    CmdStart        : BOOL ;
    CmdMov          : BOOL ;
    CmdStop         : BOOL ;
    enMoveStat      : MoveStat ;
    rSP_Vel         : REAL ;
    rSP_Acc         : REAL ;
    rSP_Dec         : REAL ;
    rSP_Distance    : REAL ;
    CmdExeMov       : BOOL ;
    CmdExeStop      : BOOL ;
    CmdSynchroOff   : BOOL ;
    CmdSynchroOn    : BOOL ;
    iStep           : INT ;
    uiiMaster       : UDINT ;
    uiMasterParID   : UINT ;
    rOverrideAcc    : REAL ;
    bSynchroOkSlavA : ARRAY [0..15]OF BOOL ;
    bTest_          : ARRAY [0..9]OF BOOL ;
    iTest_          : ARRAY [0..9]OF INT ;
    rTest_          : ARRAY [0..9]OF REAL ;
  END_STRUCT;

  CycGen : STRUCT
    bSCyc           : BOOL ;
    bFCyc           : BOOL ;
    bCyc            : BOOL ;
    bCycFail        : BOOL ;
    iStep           : INT ;
    bModTest        : BOOL ;
    bTestOn         : BOOL ;
    bTest_          : ARRAY [0..14]OF BOOL ;
    iTest_          : ARRAY [0..14]OF INT ;
    rTest_          : ARRAY [0..14]OF REAL ;
  END_STRUCT;

  CycHMPerf : STRUCT
    bSCyc           : BOOL ;
    bFCyc           : BOOL ;
    bCyc            : BOOL ;
    bCycFail        : BOOL ;
    iStep           : INT ;
    bModTest        : BOOL ;
    bTestOn         : BOOL ;
    rSP_Vel         : REAL ;
    rSP_Acc         : REAL ;
    rSP_Dec         : REAL ;
    bSlowRot_OK     : BOOL ;
    bSynchro_OK     : BOOL ;
    Cmd_SynchroOn   : BOOL ;
    Cmd_SynchroOff  : BOOL ;
    Cmd_SlowRot     : BOOL ;
    Cmd_Stop        : BOOL ;
    Cmd_EnableAxis  : BOOL ;
    bSelProd        : BOOL ;
    bStopReq        : BOOL ; (*Stop Hot Micro Perfo unit request*)
    bFaultCond      : BOOL ; (*Fault condition*)
    bStopCond       : BOOL ; (*Stop condition*)
    bSlowRotCond    : BOOL ;
    bTest_          : ARRAY [0..14]OF BOOL ;
    iTest_          : ARRAY [0..14]OF INT ;
    rTest_          : ARRAY [0..14]OF REAL ;
  END_STRUCT;

  stCycAxis : STRUCT
    CycManTimSet : CycManTimSet ;
  END_STRUCT;
END_TYPE
```

### Data object Logical/Error_Eng (Ett)

- Error_Eng.ett (not shown)

### Program Logical/HMI/BackUp (IEC)
